REGION Network 59: Magazine Z-Axis Brake Test Error
   RUNG wire#powerrail
      { S7_Templates := "SrcType := Int" } GE_Contact(in1 := "Unit1.Em5.ControlNodes".cm.brakeTest.magazine.monitoring."step", in2 := 5)
      { S7_Templates := "SrcType := Int" } LE_Contact(in1 := "Unit1.Em5.ControlNodes".cm.brakeTest.magazine.monitoring."step", in2 := 30)
      { S7_Templates := "time_type := Time" } #statTonTimer[60].TON(pt := T#10s, et =>)
      wire#w1
      Coil( "Unit1.Em5.ControlNodes".cm.brakeTest.magazine.monitoring.error )
      R_Coil( "Unit1.Em5.ControlNodes".cm.brakeTest.magazine.monitoring.busy )
      R_Coil( "Unit1.Em5.ControlNodes".cm.brakeTest.magazine.commands.axisReset )
   END_RUNG
   RUNG wire#powerrail
      Contact( "Unit1.Em5.ControlNodes".cm.brakeTest.magazine.monitoring.error )
      I_Contact( #statUnitStatus.acknowledgeActive )
   END_RUNG wire#w1
   RUNG wire#powerrail
      Contact( "Unit1.Em5.ControlNodes".cm.brakeTest.magazine.monitoring.busy )
      wire#w2
      P_Trig( #statPulse[62] )
      S_Coil( "Unit1.Em5.Config".cmMagazineAxisZ.disableAlarms )
   END_RUNG
   RUNG wire#w2
      Not()
      P_Trig( #statPulse[63] )
      R_Coil( "Unit1.Em5.Config".cmMagazineAxisZ.disableAlarms )
   END_RUNG
   // the same network as SCL:
   #statTonTimer[60].TON(IN := ("Unit1.Em5.ControlNodes".cm.brakeTest.magazine.monitoring."step" >= 5) AND ("Unit1.Em5.ControlNodes".cm.brakeTest.magazine.monitoring."step" <= 30),
                         PT := T#10s);
   "Unit1.Em5.ControlNodes".cm.brakeTest.magazine.monitoring.error := #statTonTimer[60].Q OR ("Unit1.Em5.ControlNodes".cm.brakeTest.magazine.monitoring.error AND NOT #statUnitStatus.acknowledgeActive);
   IF "Unit1.Em5.ControlNodes".cm.brakeTest.magazine.monitoring.error THEN
       "Unit1.Em5.ControlNodes".cm.brakeTest.magazine.monitoring.busy := FALSE;
       "Unit1.Em5.ControlNodes".cm.brakeTest.magazine.commands.axisReset := FALSE;
   END_IF;
   #_w1 := "Unit1.Em5.ControlNodes".cm.brakeTest.magazine.monitoring.busy AND NOT #statPulse[62];   // rising edge
   #statPulse[62] := "Unit1.Em5.ControlNodes".cm.brakeTest.magazine.monitoring.busy;
   IF #_w1 THEN "Unit1.Em5.Config".cmMagazineAxisZ.disableAlarms := TRUE; END_IF;
   #_w2 := NOT "Unit1.Em5.ControlNodes".cm.brakeTest.magazine.monitoring.busy AND NOT #statPulse[63];   // rising edge
   #statPulse[63] := NOT "Unit1.Em5.ControlNodes".cm.brakeTest.magazine.monitoring.busy;
   IF #_w2 THEN "Unit1.Em5.Config".cmMagazineAxisZ.disableAlarms := FALSE; END_IF;
END_REGION

REGION Network 60: Magazine Z-Axis Brake Test Initialize
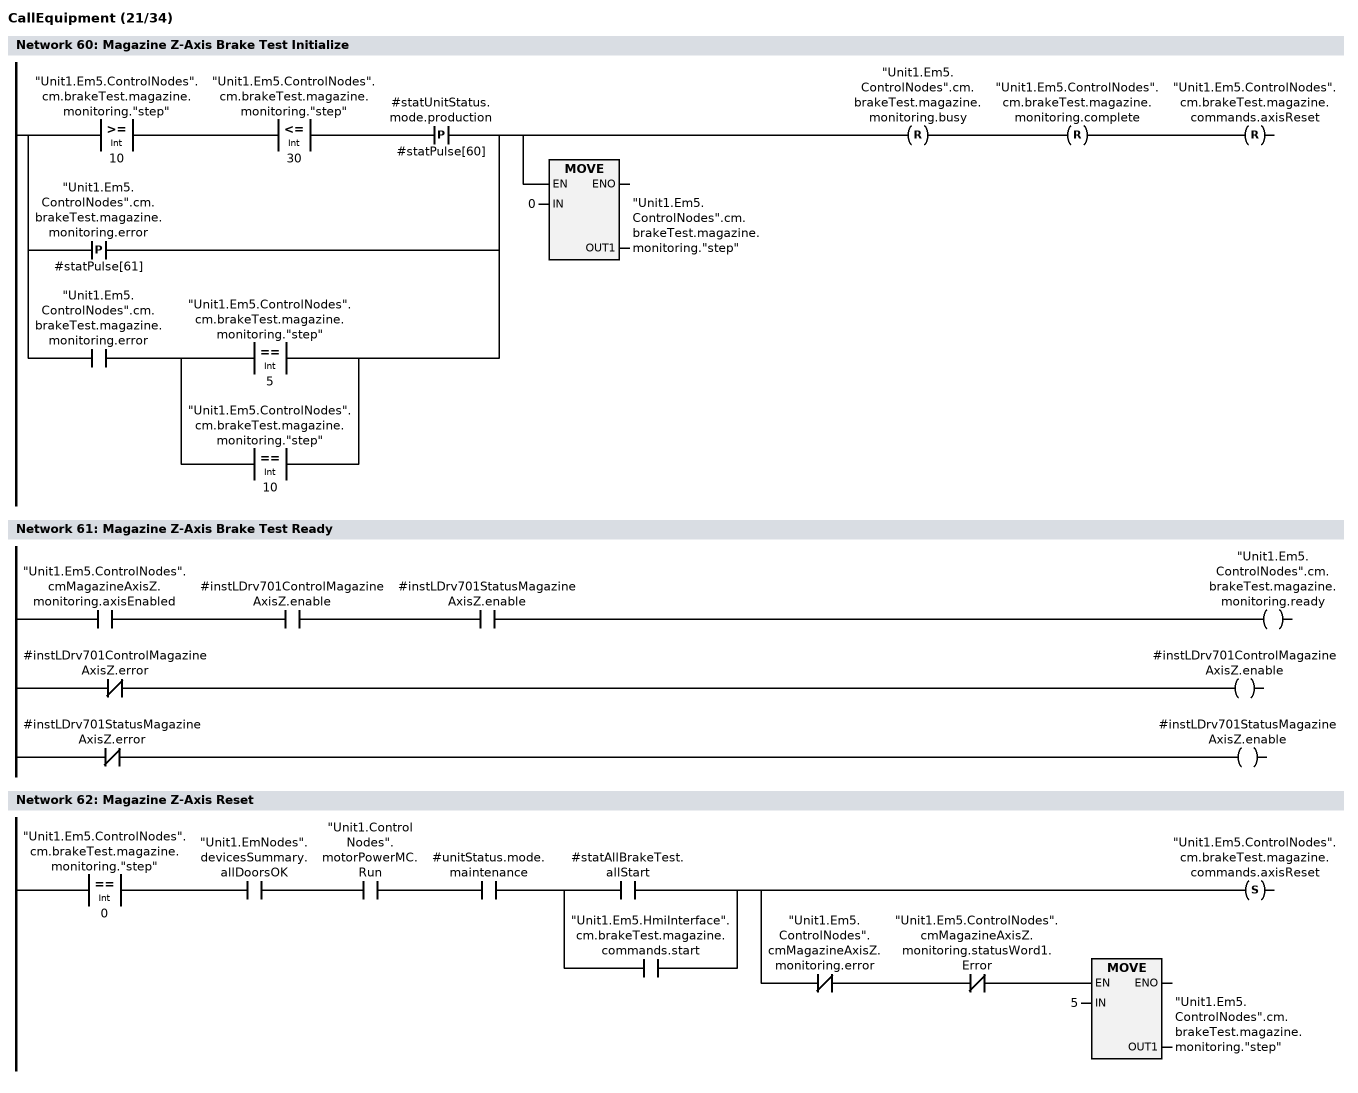
   RUNG wire#powerrail
      { S7_Templates := "SrcType := Int" } GE_Contact(in1 := "Unit1.Em5.ControlNodes".cm.brakeTest.magazine.monitoring."step", in2 := 10)
      { S7_Templates := "SrcType := Int" } LE_Contact(in1 := "Unit1.Em5.ControlNodes".cm.brakeTest.magazine.monitoring."step", in2 := 30)
      P_Contact(operand := #statUnitStatus.mode.production, bit := #statPulse[60])
      wire#w1
      R_Coil( "Unit1.Em5.ControlNodes".cm.brakeTest.magazine.monitoring.busy )
      R_Coil( "Unit1.Em5.ControlNodes".cm.brakeTest.magazine.monitoring.complete )
      R_Coil( "Unit1.Em5.ControlNodes".cm.brakeTest.magazine.commands.axisReset )
   END_RUNG
   RUNG wire#powerrail
      P_Contact(operand := "Unit1.Em5.ControlNodes".cm.brakeTest.magazine.monitoring.error, bit := #statPulse[61])
   END_RUNG wire#w1
   RUNG wire#powerrail
      Contact( "Unit1.Em5.ControlNodes".cm.brakeTest.magazine.monitoring.error )
      wire#w2
      { S7_Templates := "SrcType := Int" } EQ_Contact(in1 := "Unit1.Em5.ControlNodes".cm.brakeTest.magazine.monitoring."step", in2 := 5)
   END_RUNG wire#w1
   RUNG wire#w2
      { S7_Templates := "SrcType := Int" } EQ_Contact(in1 := "Unit1.Em5.ControlNodes".cm.brakeTest.magazine.monitoring."step", in2 := 10)
   END_RUNG wire#w1
   RUNG wire#w1
      Move(in := 0, out1 => "Unit1.Em5.ControlNodes".cm.brakeTest.magazine.monitoring."step")
   END_RUNG
   // the same network as SCL:
   #_w1 := ("Unit1.Em5.ControlNodes".cm.brakeTest.magazine.monitoring."step" >= 10) AND ("Unit1.Em5.ControlNodes".cm.brakeTest.magazine.monitoring."step" <= 30) AND #statUnitStatus.mode.production AND NOT #statPulse[60];   // rising edge of #statUnitStatus.mode.production
   #statPulse[60] := #statUnitStatus.mode.production;
   #_w2 := "Unit1.Em5.ControlNodes".cm.brakeTest.magazine.monitoring.error AND NOT #statPulse[61];   // rising edge of "Unit1.Em5.ControlNodes".cm.brakeTest.magazine.monitoring.error
   #statPulse[61] := "Unit1.Em5.ControlNodes".cm.brakeTest.magazine.monitoring.error;
   IF #_w1 OR #_w2 OR ("Unit1.Em5.ControlNodes".cm.brakeTest.magazine.monitoring.error AND (("Unit1.Em5.ControlNodes".cm.brakeTest.magazine.monitoring."step" = 5) OR ("Unit1.Em5.ControlNodes".cm.brakeTest.magazine.monitoring."step" = 10))) THEN
       "Unit1.Em5.ControlNodes".cm.brakeTest.magazine.monitoring.busy := FALSE;
       "Unit1.Em5.ControlNodes".cm.brakeTest.magazine.monitoring.complete := FALSE;
       "Unit1.Em5.ControlNodes".cm.brakeTest.magazine.commands.axisReset := FALSE;
       "Unit1.Em5.ControlNodes".cm.brakeTest.magazine.monitoring."step" := 0;
   END_IF;
END_REGION

REGION Network 61: Magazine Z-Axis Brake Test Ready
   RUNG wire#powerrail
      Contact( "Unit1.Em5.ControlNodes".cmMagazineAxisZ.monitoring.axisEnabled )
      Contact( #instLDrv701ControlMagazineAxisZ.enable )
      Contact( #instLDrv701StatusMagazineAxisZ.enable )
      Coil( "Unit1.Em5.ControlNodes".cm.brakeTest.magazine.monitoring.ready )
   END_RUNG
   RUNG wire#powerrail
      I_Contact( #instLDrv701ControlMagazineAxisZ.error )
      Coil( #instLDrv701ControlMagazineAxisZ.enable )
   END_RUNG
   RUNG wire#powerrail
      I_Contact( #instLDrv701StatusMagazineAxisZ.error )
      Coil( #instLDrv701StatusMagazineAxisZ.enable )
   END_RUNG
   // the same network as SCL:
   "Unit1.Em5.ControlNodes".cm.brakeTest.magazine.monitoring.ready := "Unit1.Em5.ControlNodes".cmMagazineAxisZ.monitoring.axisEnabled AND #instLDrv701ControlMagazineAxisZ.enable AND #instLDrv701StatusMagazineAxisZ.enable;
   #instLDrv701ControlMagazineAxisZ.enable := NOT #instLDrv701ControlMagazineAxisZ.error;
   #instLDrv701StatusMagazineAxisZ.enable := NOT #instLDrv701StatusMagazineAxisZ.error;
END_REGION

REGION Network 62: Magazine Z-Axis Reset
   RUNG wire#powerrail
      { S7_Templates := "SrcType := Int" } EQ_Contact(in1 := "Unit1.Em5.ControlNodes".cm.brakeTest.magazine.monitoring."step", in2 := 0)
      Contact( "Unit1.EmNodes".devicesSummary.allDoorsOK )
      Contact( "Unit1.ControlNodes".motorPowerMC.Run )
      Contact( #unitStatus.mode.maintenance )
      wire#w1
      Contact( #statAllBrakeTest.allStart )
      wire#w2
      S_Coil( "Unit1.Em5.ControlNodes".cm.brakeTest.magazine.commands.axisReset )
   END_RUNG
   RUNG wire#w1
      Contact( "Unit1.Em5.HmiInterface".cm.brakeTest.magazine.commands.start )
   END_RUNG wire#w2
   RUNG wire#w2
      I_Contact( "Unit1.Em5.ControlNodes".cmMagazineAxisZ.monitoring.error )
      I_Contact( "Unit1.Em5.ControlNodes".cmMagazineAxisZ.monitoring.statusWord1.Error )
      Move(in := 5, out1 => "Unit1.Em5.ControlNodes".cm.brakeTest.magazine.monitoring."step")
   END_RUNG
   // the same network as SCL:
   #_w1 := ("Unit1.Em5.ControlNodes".cm.brakeTest.magazine.monitoring."step" = 0) AND "Unit1.EmNodes".devicesSummary.allDoorsOK AND "Unit1.ControlNodes".motorPowerMC.Run AND #unitStatus.mode.maintenance AND (#statAllBrakeTest.allStart OR "Unit1.Em5.HmiInterface".cm.brakeTest.magazine.commands.start);
   IF #_w1 THEN "Unit1.Em5.ControlNodes".cm.brakeTest.magazine.commands.axisReset := TRUE; END_IF;
   IF #_w1 AND NOT "Unit1.Em5.ControlNodes".cmMagazineAxisZ.monitoring.error AND NOT "Unit1.Em5.ControlNodes".cmMagazineAxisZ.monitoring.statusWord1.Error THEN
       "Unit1.Em5.ControlNodes".cm.brakeTest.magazine.monitoring."step" := 5;
   END_IF;
END_REGION

REGION Network 63: Magazine Z-Axis Brake Test Commands
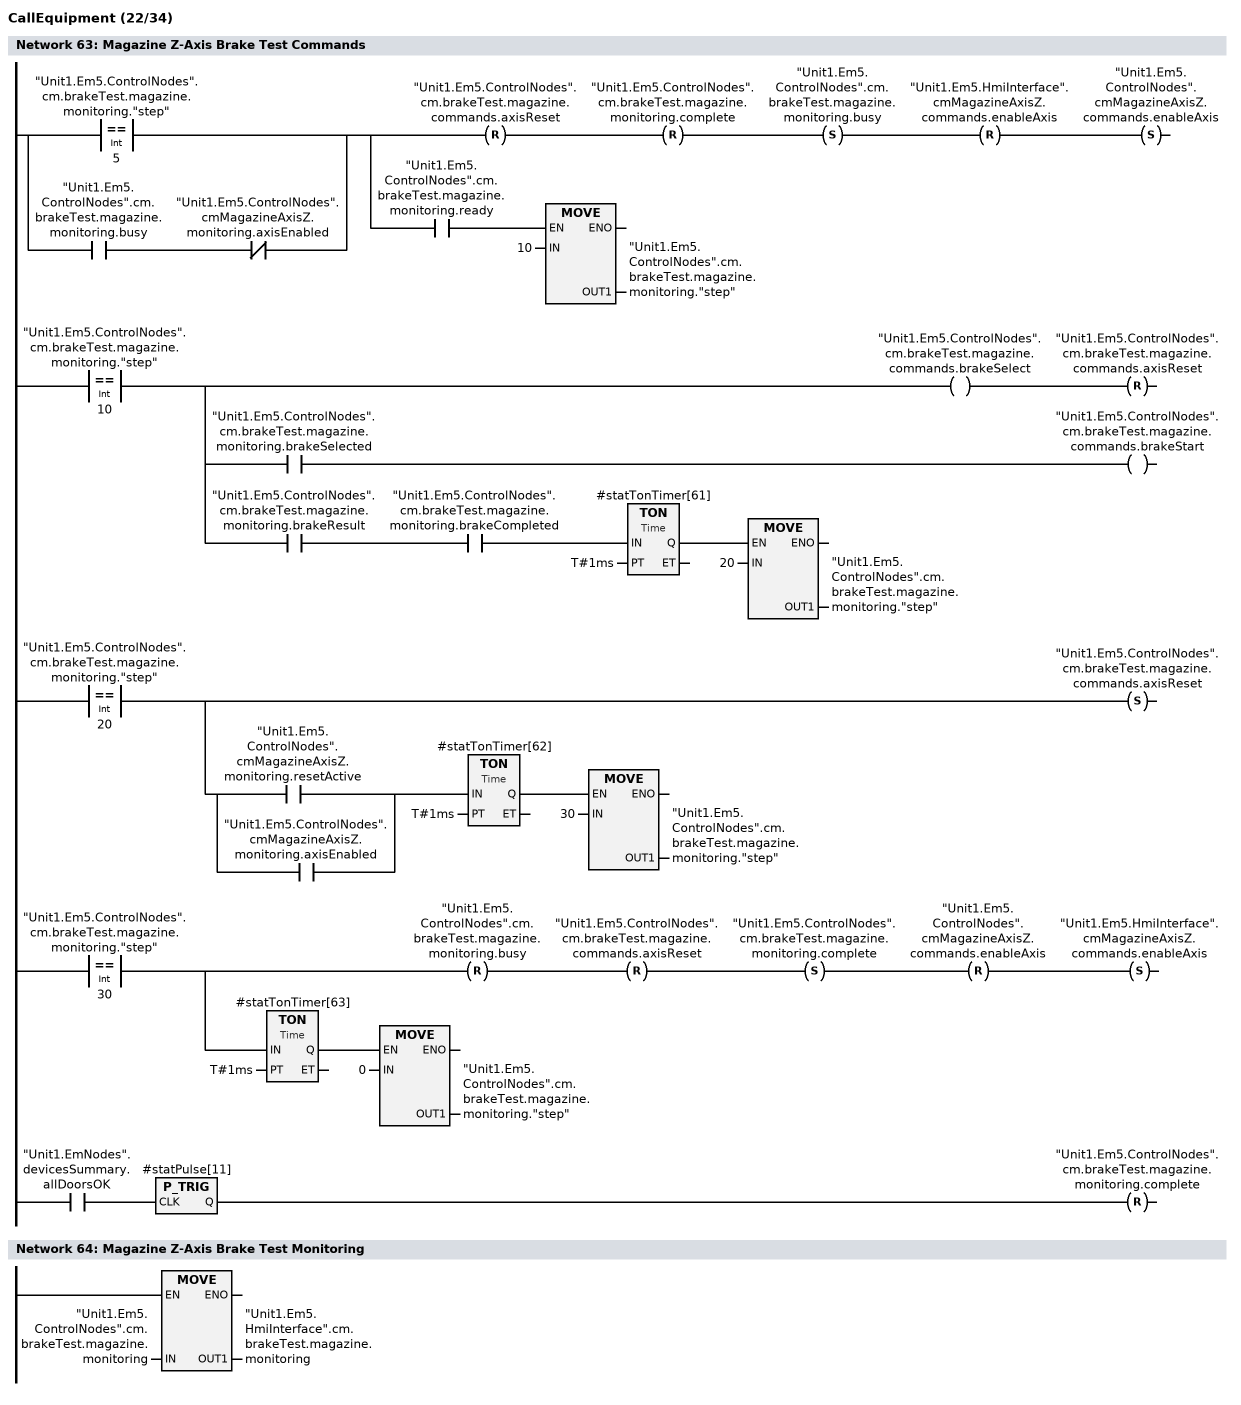
   RUNG wire#powerrail
      { S7_Templates := "SrcType := Int" } EQ_Contact(in1 := "Unit1.Em5.ControlNodes".cm.brakeTest.magazine.monitoring."step", in2 := 5)
      wire#w1
      R_Coil( "Unit1.Em5.ControlNodes".cm.brakeTest.magazine.commands.axisReset )
      R_Coil( "Unit1.Em5.ControlNodes".cm.brakeTest.magazine.monitoring.complete )
      S_Coil( "Unit1.Em5.ControlNodes".cm.brakeTest.magazine.monitoring.busy )
      R_Coil( "Unit1.Em5.HmiInterface".cmMagazineAxisZ.commands.enableAxis )
      S_Coil( "Unit1.Em5.ControlNodes".cmMagazineAxisZ.commands.enableAxis )
   END_RUNG
   RUNG wire#powerrail
      Contact( "Unit1.Em5.ControlNodes".cm.brakeTest.magazine.monitoring.busy )
      I_Contact( "Unit1.Em5.ControlNodes".cmMagazineAxisZ.monitoring.axisEnabled )
   END_RUNG wire#w1
   RUNG wire#w1
      Contact( "Unit1.Em5.ControlNodes".cm.brakeTest.magazine.monitoring.ready )
      Move(in := 10, out1 => "Unit1.Em5.ControlNodes".cm.brakeTest.magazine.monitoring."step")
   END_RUNG
   RUNG wire#powerrail
      { S7_Templates := "SrcType := Int" } EQ_Contact(in1 := "Unit1.Em5.ControlNodes".cm.brakeTest.magazine.monitoring."step", in2 := 10)
      wire#w2
      Coil( "Unit1.Em5.ControlNodes".cm.brakeTest.magazine.commands.brakeSelect )
      R_Coil( "Unit1.Em5.ControlNodes".cm.brakeTest.magazine.commands.axisReset )
   END_RUNG
   RUNG wire#w2
      Contact( "Unit1.Em5.ControlNodes".cm.brakeTest.magazine.monitoring.brakeSelected )
      Coil( "Unit1.Em5.ControlNodes".cm.brakeTest.magazine.commands.brakeStart )
   END_RUNG
   RUNG wire#w2
      Contact( "Unit1.Em5.ControlNodes".cm.brakeTest.magazine.monitoring.brakeResult )
      Contact( "Unit1.Em5.ControlNodes".cm.brakeTest.magazine.monitoring.brakeCompleted )
      { S7_Templates := "time_type := Time" } #statTonTimer[61].TON(pt := T#1ms, et =>)
      Move(in := 20, out1 => "Unit1.Em5.ControlNodes".cm.brakeTest.magazine.monitoring."step")
   END_RUNG
   RUNG wire#powerrail
      { S7_Templates := "SrcType := Int" } EQ_Contact(in1 := "Unit1.Em5.ControlNodes".cm.brakeTest.magazine.monitoring."step", in2 := 20)
      wire#w3
      S_Coil( "Unit1.Em5.ControlNodes".cm.brakeTest.magazine.commands.axisReset )
   END_RUNG
   RUNG wire#w3
      Contact( "Unit1.Em5.ControlNodes".cmMagazineAxisZ.monitoring.resetActive )
      wire#w4
      { S7_Templates := "time_type := Time" } #statTonTimer[62].TON(pt := T#1ms, et =>)
      Move(in := 30, out1 => "Unit1.Em5.ControlNodes".cm.brakeTest.magazine.monitoring."step")
   END_RUNG
   RUNG wire#w3
      Contact( "Unit1.Em5.ControlNodes".cmMagazineAxisZ.monitoring.axisEnabled )
   END_RUNG wire#w4
   RUNG wire#powerrail
      { S7_Templates := "SrcType := Int" } EQ_Contact(in1 := "Unit1.Em5.ControlNodes".cm.brakeTest.magazine.monitoring."step", in2 := 30)
      wire#w5
      R_Coil( "Unit1.Em5.ControlNodes".cm.brakeTest.magazine.monitoring.busy )
      R_Coil( "Unit1.Em5.ControlNodes".cm.brakeTest.magazine.commands.axisReset )
      S_Coil( "Unit1.Em5.ControlNodes".cm.brakeTest.magazine.monitoring.complete )
      R_Coil( "Unit1.Em5.ControlNodes".cmMagazineAxisZ.commands.enableAxis )
      S_Coil( "Unit1.Em5.HmiInterface".cmMagazineAxisZ.commands.enableAxis )
   END_RUNG
   RUNG wire#w5
      { S7_Templates := "time_type := Time" } #statTonTimer[63].TON(pt := T#1ms, et =>)
      Move(in := 0, out1 => "Unit1.Em5.ControlNodes".cm.brakeTest.magazine.monitoring."step")
   END_RUNG
   RUNG wire#powerrail
      Contact( "Unit1.EmNodes".devicesSummary.allDoorsOK )
      P_Trig( #statPulse[11] )
      R_Coil( "Unit1.Em5.ControlNodes".cm.brakeTest.magazine.monitoring.complete )
   END_RUNG
   // the same network as SCL:
   #_w1 := ("Unit1.Em5.ControlNodes".cm.brakeTest.magazine.monitoring."step" = 5) OR ("Unit1.Em5.ControlNodes".cm.brakeTest.magazine.monitoring.busy AND NOT "Unit1.Em5.ControlNodes".cmMagazineAxisZ.monitoring.axisEnabled);
   IF #_w1 THEN
       "Unit1.Em5.ControlNodes".cm.brakeTest.magazine.commands.axisReset := FALSE;
       "Unit1.Em5.ControlNodes".cm.brakeTest.magazine.monitoring.complete := FALSE;
       "Unit1.Em5.ControlNodes".cm.brakeTest.magazine.monitoring.busy := TRUE;
       "Unit1.Em5.HmiInterface".cmMagazineAxisZ.commands.enableAxis := FALSE;
       "Unit1.Em5.ControlNodes".cmMagazineAxisZ.commands.enableAxis := TRUE;
   END_IF;
   IF #_w1 AND "Unit1.Em5.ControlNodes".cm.brakeTest.magazine.monitoring.ready THEN
       "Unit1.Em5.ControlNodes".cm.brakeTest.magazine.monitoring."step" := 10;
   END_IF;
   "Unit1.Em5.ControlNodes".cm.brakeTest.magazine.commands.brakeSelect := "Unit1.Em5.ControlNodes".cm.brakeTest.magazine.monitoring."step" = 10;
   IF "Unit1.Em5.ControlNodes".cm.brakeTest.magazine.commands.brakeSelect THEN
       "Unit1.Em5.ControlNodes".cm.brakeTest.magazine.commands.axisReset := FALSE;
   END_IF;
   "Unit1.Em5.ControlNodes".cm.brakeTest.magazine.commands.brakeStart := "Unit1.Em5.ControlNodes".cm.brakeTest.magazine.commands.brakeSelect AND "Unit1.Em5.ControlNodes".cm.brakeTest.magazine.monitoring.brakeSelected;
   #statTonTimer[61].TON(IN := "Unit1.Em5.ControlNodes".cm.brakeTest.magazine.commands.brakeSelect AND "Unit1.Em5.ControlNodes".cm.brakeTest.magazine.monitoring.brakeResult AND "Unit1.Em5.ControlNodes".cm.brakeTest.magazine.monitoring.brakeCompleted,
                         PT := T#1ms);
   IF #statTonTimer[61].Q THEN
       "Unit1.Em5.ControlNodes".cm.brakeTest.magazine.monitoring."step" := 20;
   END_IF;
   #_w2 := "Unit1.Em5.ControlNodes".cm.brakeTest.magazine.monitoring."step" = 20;
   IF #_w2 THEN "Unit1.Em5.ControlNodes".cm.brakeTest.magazine.commands.axisReset := TRUE; END_IF;
   #statTonTimer[62].TON(IN := #_w2 AND ("Unit1.Em5.ControlNodes".cmMagazineAxisZ.monitoring.resetActive OR "Unit1.Em5.ControlNodes".cmMagazineAxisZ.monitoring.axisEnabled),
                         PT := T#1ms);
   IF #statTonTimer[62].Q THEN
       "Unit1.Em5.ControlNodes".cm.brakeTest.magazine.monitoring."step" := 30;
   END_IF;
   #_w3 := "Unit1.Em5.ControlNodes".cm.brakeTest.magazine.monitoring."step" = 30;
   IF #_w3 THEN
       "Unit1.Em5.ControlNodes".cm.brakeTest.magazine.monitoring.busy := FALSE;
       "Unit1.Em5.ControlNodes".cm.brakeTest.magazine.commands.axisReset := FALSE;
       "Unit1.Em5.ControlNodes".cm.brakeTest.magazine.monitoring.complete := TRUE;
       "Unit1.Em5.ControlNodes".cmMagazineAxisZ.commands.enableAxis := FALSE;
       "Unit1.Em5.HmiInterface".cmMagazineAxisZ.commands.enableAxis := TRUE;
   END_IF;
   #statTonTimer[63].TON(IN := #_w3, PT := T#1ms);
   IF #statTonTimer[63].Q THEN "Unit1.Em5.ControlNodes".cm.brakeTest.magazine.monitoring."step" := 0; END_IF;
   #_w4 := "Unit1.EmNodes".devicesSummary.allDoorsOK AND NOT #statPulse[11];   // rising edge
   #statPulse[11] := "Unit1.EmNodes".devicesSummary.allDoorsOK;
   IF #_w4 THEN "Unit1.Em5.ControlNodes".cm.brakeTest.magazine.monitoring.complete := FALSE; END_IF;
END_REGION

REGION Network 64: Magazine Z-Axis Brake Test Monitoring
   RUNG wire#powerrail
      Move(in := "Unit1.Em5.ControlNodes".cm.brakeTest.magazine.monitoring, out1 => "Unit1.Em5.HmiInterface".cm.brakeTest.magazine.monitoring)
   END_RUNG
   // the same network as SCL:
   "Unit1.Em5.HmiInterface".cm.brakeTest.magazine.monitoring := "Unit1.Em5.ControlNodes".cm.brakeTest.magazine.monitoring;
END_REGION

REGION Network 65: Call Magazine Z-Axis Telegram 701
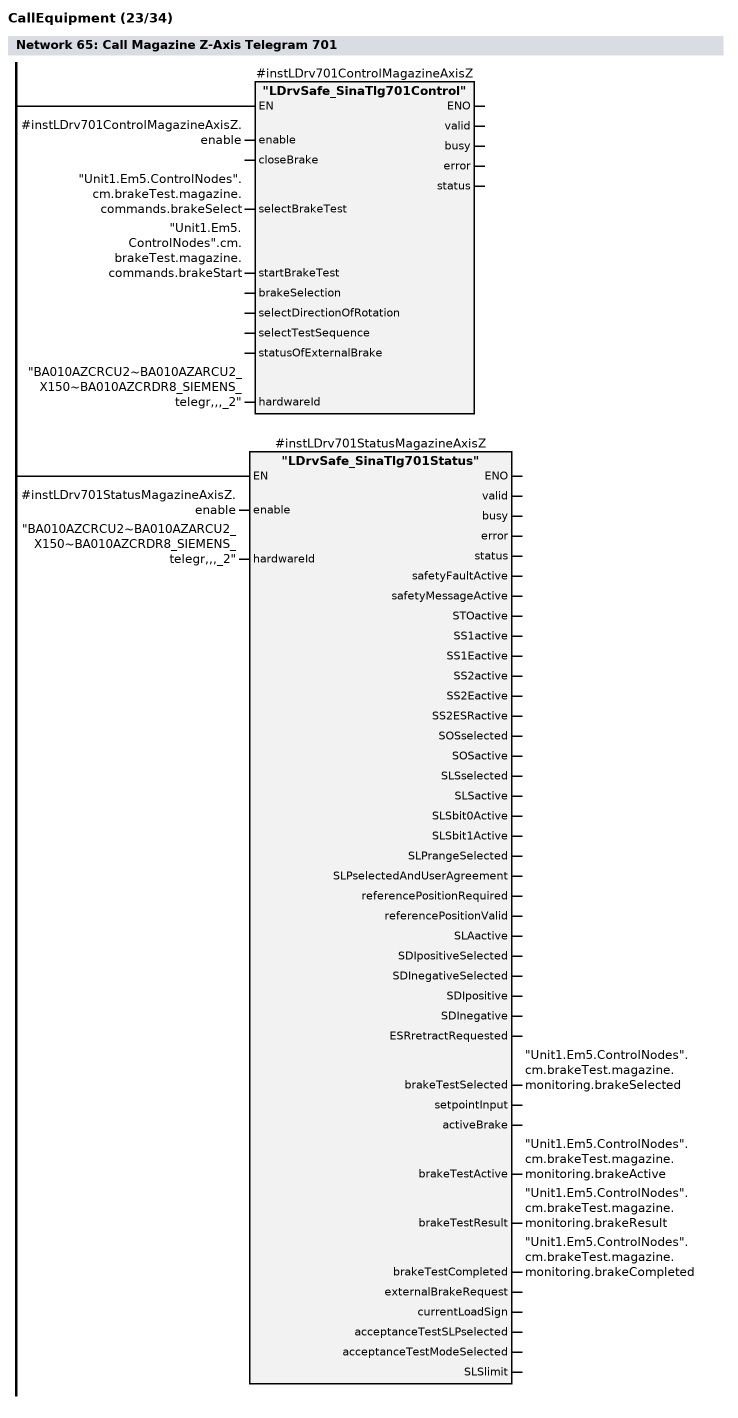
   RUNG wire#powerrail
      #instLDrv701ControlMagazineAxisZ(enable := #instLDrv701ControlMagazineAxisZ.enable, closeBrake :=, selectBrakeTest := "Unit1.Em5.ControlNodes".cm.brakeTest.magazine.commands.brakeSelect, startBrakeTest := "Unit1.Em5.ControlNodes".cm.brakeTest.magazine.commands.brakeStart, brakeSelection :=, selectDirectionOfRotation :=, selectTestSequence :=, statusOfExternalBrake :=, hardwareId := "BA010AZCRCU2~BA010AZARCU2_X150~BA010AZCRDR8_SIEMENS_telegr,,,_2", valid =>, busy =>, error =>, status =>)
   END_RUNG
   RUNG wire#powerrail
      #instLDrv701StatusMagazineAxisZ(enable := #instLDrv701StatusMagazineAxisZ.enable, hardwareId := "BA010AZCRCU2~BA010AZARCU2_X150~BA010AZCRDR8_SIEMENS_telegr,,,_2", valid =>, busy =>, error =>, status =>, safetyFaultActive =>, safetyMessageActive =>, STOactive =>, SS1active =>, SS1Eactive =>, SS2active =>, SS2Eactive =>, SS2ESRactive =>, SOSselected =>, SOSactive =>, SLSselected =>, SLSactive =>, SLSbit0Active =>, SLSbit1Active =>, SLPrangeSelected =>, SLPselectedAndUserAgreement =>, referencePositionRequired =>, referencePositionValid =>, SLAactive =>, SDIpositiveSelected =>, SDInegativeSelected =>, SDIpositive =>, SDInegative =>, ESRretractRequested =>, brakeTestSelected => "Unit1.Em5.ControlNodes".cm.brakeTest.magazine.monitoring.brakeSelected, setpointInput =>, activeBrake =>, brakeTestActive => "Unit1.Em5.ControlNodes".cm.brakeTest.magazine.monitoring.brakeActive, brakeTestResult => "Unit1.Em5.ControlNodes".cm.brakeTest.magazine.monitoring.brakeResult, brakeTestCompleted => "Unit1.Em5.ControlNodes".cm.brakeTest.magazine.monitoring.brakeCompleted, externalBrakeRequest =>, currentLoadSign =>, acceptanceTestSLPselected =>, acceptanceTestModeSelected =>, SLSlimit =>)
   END_RUNG
   // the same network as SCL:
   #instLDrv701ControlMagazineAxisZ(enable := #instLDrv701ControlMagazineAxisZ.enable,   // "LDrvSafe_SinaTlg701Control"
                           selectBrakeTest := "Unit1.Em5.ControlNodes".cm.brakeTest.magazine.commands.brakeSelect,
                           startBrakeTest := "Unit1.Em5.ControlNodes".cm.brakeTest.magazine.commands.brakeStart,
                           hardwareId := "BA010AZCRCU2~BA010AZARCU2_X150~BA010AZCRDR8_SIEMENS_telegr,,,_2");
   #instLDrv701StatusMagazineAxisZ(enable := #instLDrv701StatusMagazineAxisZ.enable,   // "LDrvSafe_SinaTlg701Status"
                           hardwareId := "BA010AZCRCU2~BA010AZARCU2_X150~BA010AZCRDR8_SIEMENS_telegr,,,_2",
                           brakeTestSelected => "Unit1.Em5.ControlNodes".cm.brakeTest.magazine.monitoring.brakeSelected,
                           brakeTestActive => "Unit1.Em5.ControlNodes".cm.brakeTest.magazine.monitoring.brakeActive,
                           brakeTestResult => "Unit1.Em5.ControlNodes".cm.brakeTest.magazine.monitoring.brakeResult,
                           brakeTestCompleted => "Unit1.Em5.ControlNodes".cm.brakeTest.magazine.monitoring.brakeCompleted);
END_REGION

REGION Network 67: ******************** Control Modules (TwoWayActuator) ********************
   // Call control modules that are actuators after the em logic (jobs and sequence), so that the latest commands are applied to the actuators.
END_REGION

REGION Network 68: Reset CMS
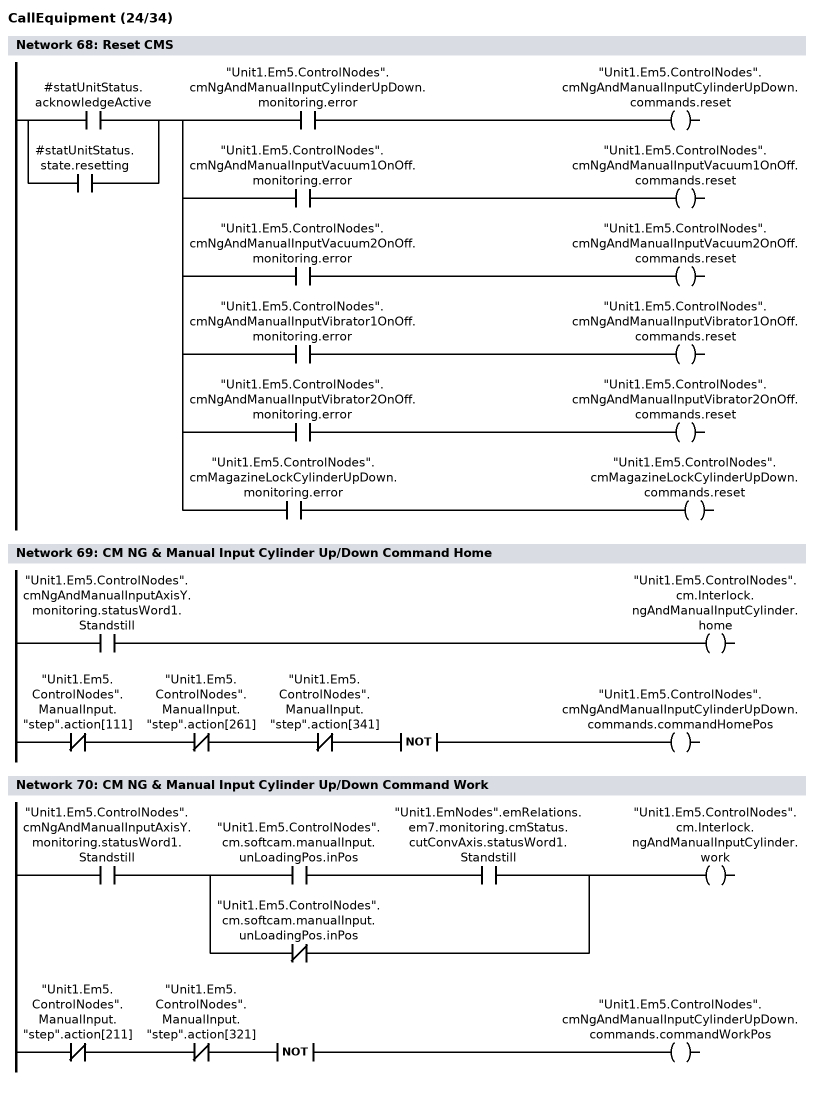
   RUNG wire#powerrail
      Contact( #statUnitStatus.acknowledgeActive )
      wire#w1
      Contact( "Unit1.Em5.ControlNodes".cmNgAndManualInputCylinderUpDown.monitoring.error )
      Coil( "Unit1.Em5.ControlNodes".cmNgAndManualInputCylinderUpDown.commands.reset )
   END_RUNG
   RUNG wire#powerrail
      Contact( #statUnitStatus.state.resetting )
   END_RUNG wire#w1
   RUNG wire#w1
      Contact( "Unit1.Em5.ControlNodes".cmNgAndManualInputVacuum1OnOff.monitoring.error )
      Coil( "Unit1.Em5.ControlNodes".cmNgAndManualInputVacuum1OnOff.commands.reset )
   END_RUNG
   RUNG wire#w1
      Contact( "Unit1.Em5.ControlNodes".cmNgAndManualInputVacuum2OnOff.monitoring.error )
      Coil( "Unit1.Em5.ControlNodes".cmNgAndManualInputVacuum2OnOff.commands.reset )
   END_RUNG
   RUNG wire#w1
      Contact( "Unit1.Em5.ControlNodes".cmNgAndManualInputVibrator1OnOff.monitoring.error )
      Coil( "Unit1.Em5.ControlNodes".cmNgAndManualInputVibrator1OnOff.commands.reset )
   END_RUNG
   RUNG wire#w1
      Contact( "Unit1.Em5.ControlNodes".cmNgAndManualInputVibrator2OnOff.monitoring.error )
      Coil( "Unit1.Em5.ControlNodes".cmNgAndManualInputVibrator2OnOff.commands.reset )
   END_RUNG
   RUNG wire#w1
      Contact( "Unit1.Em5.ControlNodes".cmMagazineLockCylinderUpDown.monitoring.error )
      Coil( "Unit1.Em5.ControlNodes".cmMagazineLockCylinderUpDown.commands.reset )
   END_RUNG
   // the same network as SCL:
   #_w1 := #statUnitStatus.acknowledgeActive OR #statUnitStatus.state.resetting;
   "Unit1.Em5.ControlNodes".cmNgAndManualInputCylinderUpDown.commands.reset := #_w1 AND "Unit1.Em5.ControlNodes".cmNgAndManualInputCylinderUpDown.monitoring.error;
   "Unit1.Em5.ControlNodes".cmNgAndManualInputVacuum1OnOff.commands.reset := #_w1 AND "Unit1.Em5.ControlNodes".cmNgAndManualInputVacuum1OnOff.monitoring.error;
   "Unit1.Em5.ControlNodes".cmNgAndManualInputVacuum2OnOff.commands.reset := #_w1 AND "Unit1.Em5.ControlNodes".cmNgAndManualInputVacuum2OnOff.monitoring.error;
   "Unit1.Em5.ControlNodes".cmNgAndManualInputVibrator1OnOff.commands.reset := #_w1 AND "Unit1.Em5.ControlNodes".cmNgAndManualInputVibrator1OnOff.monitoring.error;
   "Unit1.Em5.ControlNodes".cmNgAndManualInputVibrator2OnOff.commands.reset := #_w1 AND "Unit1.Em5.ControlNodes".cmNgAndManualInputVibrator2OnOff.monitoring.error;
   "Unit1.Em5.ControlNodes".cmMagazineLockCylinderUpDown.commands.reset := #_w1 AND "Unit1.Em5.ControlNodes".cmMagazineLockCylinderUpDown.monitoring.error;
END_REGION

REGION Network 69: CM NG & Manual Input Cylinder Up/Down Command Home
   RUNG wire#powerrail
      Contact( "Unit1.Em5.ControlNodes".cmNgAndManualInputAxisY.monitoring.statusWord1.Standstill )
      Coil( "Unit1.Em5.ControlNodes".cm.Interlock.ngAndManualInputCylinder.home )
   END_RUNG
   RUNG wire#powerrail
      I_Contact( "Unit1.Em5.ControlNodes".ManualInput."step".action[111] )
      I_Contact( "Unit1.Em5.ControlNodes".ManualInput."step".action[261] )
      I_Contact( "Unit1.Em5.ControlNodes".ManualInput."step".action[341] )
      Not()
      Coil( "Unit1.Em5.ControlNodes".cmNgAndManualInputCylinderUpDown.commands.commandHomePos )
   END_RUNG
   // the same network as SCL:
   "Unit1.Em5.ControlNodes".cm.Interlock.ngAndManualInputCylinder.home := "Unit1.Em5.ControlNodes".cmNgAndManualInputAxisY.monitoring.statusWord1.Standstill;
   "Unit1.Em5.ControlNodes".cmNgAndManualInputCylinderUpDown.commands.commandHomePos := NOT (NOT "Unit1.Em5.ControlNodes".ManualInput."step".action[111] AND NOT "Unit1.Em5.ControlNodes".ManualInput."step".action[261] AND NOT "Unit1.Em5.ControlNodes".ManualInput."step".action[341]);
END_REGION

REGION Network 70: CM NG & Manual Input Cylinder Up/Down Command Work
   RUNG wire#powerrail
      Contact( "Unit1.Em5.ControlNodes".cmNgAndManualInputAxisY.monitoring.statusWord1.Standstill )
      wire#w1
      Contact( "Unit1.Em5.ControlNodes".cm.softcam.manualInput.unLoadingPos.inPos )
      Contact( "Unit1.EmNodes".emRelations.em7.monitoring.cmStatus.cutConvAxis.statusWord1.Standstill )
      wire#w2
      Coil( "Unit1.Em5.ControlNodes".cm.Interlock.ngAndManualInputCylinder.work )
   END_RUNG
   RUNG wire#w1
      I_Contact( "Unit1.Em5.ControlNodes".cm.softcam.manualInput.unLoadingPos.inPos )
   END_RUNG wire#w2
   RUNG wire#powerrail
      I_Contact( "Unit1.Em5.ControlNodes".ManualInput."step".action[211] )
      I_Contact( "Unit1.Em5.ControlNodes".ManualInput."step".action[321] )
      Not()
      Coil( "Unit1.Em5.ControlNodes".cmNgAndManualInputCylinderUpDown.commands.commandWorkPos )
   END_RUNG
   // the same network as SCL:
   "Unit1.Em5.ControlNodes".cm.Interlock.ngAndManualInputCylinder.work := "Unit1.Em5.ControlNodes".cmNgAndManualInputAxisY.monitoring.statusWord1.Standstill AND (("Unit1.Em5.ControlNodes".cm.softcam.manualInput.unLoadingPos.inPos AND "Unit1.EmNodes".emRelations.em7.monitoring.cmStatus.cutConvAxis.statusWord1.Standstill) OR NOT "Unit1.Em5.ControlNodes".cm.softcam.manualInput.unLoadingPos.inPos);
   "Unit1.Em5.ControlNodes".cmNgAndManualInputCylinderUpDown.commands.commandWorkPos := NOT (NOT "Unit1.Em5.ControlNodes".ManualInput."step".action[211] AND NOT "Unit1.Em5.ControlNodes".ManualInput."step".action[321]);
END_REGION

REGION Network 71: Call CM NG & Manual Input Cylinder Up/Down (LBC_TwoWayActuator)
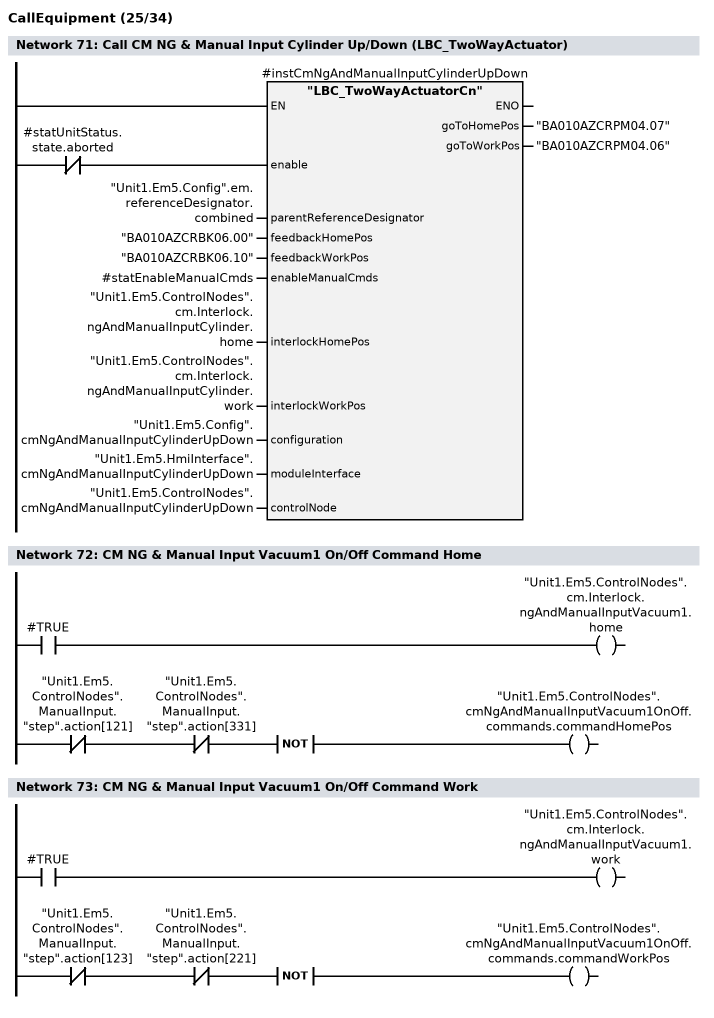
   RUNG wire#powerrail
      #instCmNgAndManualInputCylinderUpDown(enable := wire#w1, parentReferenceDesignator := "Unit1.Em5.Config".em.referenceDesignator.combined, feedbackHomePos := "BA010AZCRBK06.00", feedbackWorkPos := "BA010AZCRBK06.10", enableManualCmds := #statEnableManualCmds, interlockHomePos := "Unit1.Em5.ControlNodes".cm.Interlock.ngAndManualInputCylinder.home, interlockWorkPos := "Unit1.Em5.ControlNodes".cm.Interlock.ngAndManualInputCylinder.work, configuration := "Unit1.Em5.Config".cmNgAndManualInputCylinderUpDown, moduleInterface := "Unit1.Em5.HmiInterface".cmNgAndManualInputCylinderUpDown, controlNode := "Unit1.Em5.ControlNodes".cmNgAndManualInputCylinderUpDown, goToHomePos => "BA010AZCRPM04.07", goToWorkPos => "BA010AZCRPM04.06")
   END_RUNG
   RUNG wire#powerrail
      I_Contact( #statUnitStatus.state.aborted )
   END_RUNG wire#w1
   // the same network as SCL:
   #instCmNgAndManualInputCylinderUpDown(enable := NOT #statUnitStatus.state.aborted,   // "LBC_TwoWayActuatorCn"
                           parentReferenceDesignator := "Unit1.Em5.Config".em.referenceDesignator.combined,
                           feedbackHomePos := "BA010AZCRBK06.00",
                           feedbackWorkPos := "BA010AZCRBK06.10",
                           enableManualCmds := #statEnableManualCmds,
                           interlockHomePos := "Unit1.Em5.ControlNodes".cm.Interlock.ngAndManualInputCylinder.home,
                           interlockWorkPos := "Unit1.Em5.ControlNodes".cm.Interlock.ngAndManualInputCylinder.work,
                           configuration := "Unit1.Em5.Config".cmNgAndManualInputCylinderUpDown,
                           moduleInterface := "Unit1.Em5.HmiInterface".cmNgAndManualInputCylinderUpDown,
                           controlNode := "Unit1.Em5.ControlNodes".cmNgAndManualInputCylinderUpDown,
                           goToHomePos => "BA010AZCRPM04.07",
                           goToWorkPos => "BA010AZCRPM04.06");
END_REGION

REGION Network 72: CM NG & Manual Input Vacuum1 On/Off Command Home
   RUNG wire#powerrail
      Contact( #TRUE )
      Coil( "Unit1.Em5.ControlNodes".cm.Interlock.ngAndManualInputVacuum1.home )
   END_RUNG
   RUNG wire#powerrail
      I_Contact( "Unit1.Em5.ControlNodes".ManualInput."step".action[121] )
      I_Contact( "Unit1.Em5.ControlNodes".ManualInput."step".action[331] )
      Not()
      Coil( "Unit1.Em5.ControlNodes".cmNgAndManualInputVacuum1OnOff.commands.commandHomePos )
   END_RUNG
   // the same network as SCL:
   "Unit1.Em5.ControlNodes".cm.Interlock.ngAndManualInputVacuum1.home := #TRUE;
   "Unit1.Em5.ControlNodes".cmNgAndManualInputVacuum1OnOff.commands.commandHomePos := NOT (NOT "Unit1.Em5.ControlNodes".ManualInput."step".action[121] AND NOT "Unit1.Em5.ControlNodes".ManualInput."step".action[331]);
END_REGION

REGION Network 73: CM NG & Manual Input Vacuum1 On/Off Command Work
   RUNG wire#powerrail
      Contact( #TRUE )
      Coil( "Unit1.Em5.ControlNodes".cm.Interlock.ngAndManualInputVacuum1.work )
   END_RUNG
   RUNG wire#powerrail
      I_Contact( "Unit1.Em5.ControlNodes".ManualInput."step".action[123] )
      I_Contact( "Unit1.Em5.ControlNodes".ManualInput."step".action[221] )
      Not()
      Coil( "Unit1.Em5.ControlNodes".cmNgAndManualInputVacuum1OnOff.commands.commandWorkPos )
   END_RUNG
   // the same network as SCL:
   "Unit1.Em5.ControlNodes".cm.Interlock.ngAndManualInputVacuum1.work := #TRUE;
   "Unit1.Em5.ControlNodes".cmNgAndManualInputVacuum1OnOff.commands.commandWorkPos := NOT (NOT "Unit1.Em5.ControlNodes".ManualInput."step".action[123] AND NOT "Unit1.Em5.ControlNodes".ManualInput."step".action[221]);
END_REGION

REGION Network 74: Call CM NG & Manual Input Vacuum1 On/Off (LBC_TwoWayActuator)
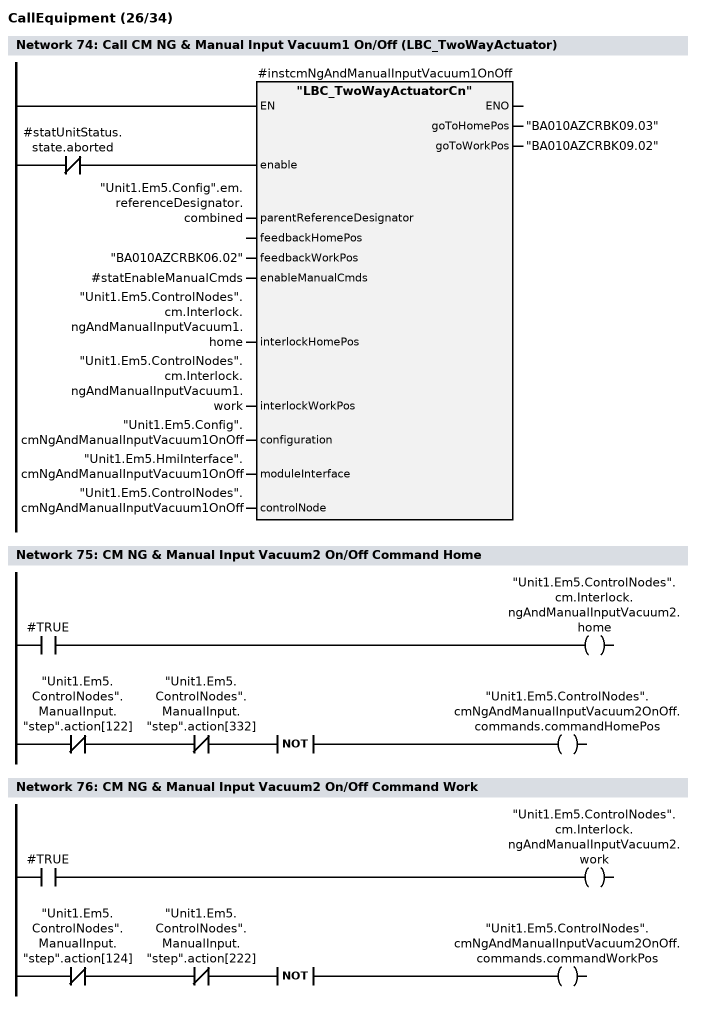
   RUNG wire#powerrail
      #instcmNgAndManualInputVacuum1OnOff(enable := wire#w1, parentReferenceDesignator := "Unit1.Em5.Config".em.referenceDesignator.combined, feedbackHomePos :=, feedbackWorkPos := "BA010AZCRBK06.02", enableManualCmds := #statEnableManualCmds, interlockHomePos := "Unit1.Em5.ControlNodes".cm.Interlock.ngAndManualInputVacuum1.home, interlockWorkPos := "Unit1.Em5.ControlNodes".cm.Interlock.ngAndManualInputVacuum1.work, configuration := "Unit1.Em5.Config".cmNgAndManualInputVacuum1OnOff, moduleInterface := "Unit1.Em5.HmiInterface".cmNgAndManualInputVacuum1OnOff, controlNode := "Unit1.Em5.ControlNodes".cmNgAndManualInputVacuum1OnOff, goToHomePos => "BA010AZCRBK09.03", goToWorkPos => "BA010AZCRBK09.02")
   END_RUNG
   RUNG wire#powerrail
      I_Contact( #statUnitStatus.state.aborted )
   END_RUNG wire#w1
   // the same network as SCL:
   #instcmNgAndManualInputVacuum1OnOff(enable := NOT #statUnitStatus.state.aborted,   // "LBC_TwoWayActuatorCn"
                           parentReferenceDesignator := "Unit1.Em5.Config".em.referenceDesignator.combined,
                           feedbackWorkPos := "BA010AZCRBK06.02",
                           enableManualCmds := #statEnableManualCmds,
                           interlockHomePos := "Unit1.Em5.ControlNodes".cm.Interlock.ngAndManualInputVacuum1.home,
                           interlockWorkPos := "Unit1.Em5.ControlNodes".cm.Interlock.ngAndManualInputVacuum1.work,
                           configuration := "Unit1.Em5.Config".cmNgAndManualInputVacuum1OnOff,
                           moduleInterface := "Unit1.Em5.HmiInterface".cmNgAndManualInputVacuum1OnOff,
                           controlNode := "Unit1.Em5.ControlNodes".cmNgAndManualInputVacuum1OnOff,
                           goToHomePos => "BA010AZCRBK09.03",
                           goToWorkPos => "BA010AZCRBK09.02");
END_REGION

REGION Network 75: CM NG & Manual Input Vacuum2 On/Off Command Home
   RUNG wire#powerrail
      Contact( #TRUE )
      Coil( "Unit1.Em5.ControlNodes".cm.Interlock.ngAndManualInputVacuum2.home )
   END_RUNG
   RUNG wire#powerrail
      I_Contact( "Unit1.Em5.ControlNodes".ManualInput."step".action[122] )
      I_Contact( "Unit1.Em5.ControlNodes".ManualInput."step".action[332] )
      Not()
      Coil( "Unit1.Em5.ControlNodes".cmNgAndManualInputVacuum2OnOff.commands.commandHomePos )
   END_RUNG
   // the same network as SCL:
   "Unit1.Em5.ControlNodes".cm.Interlock.ngAndManualInputVacuum2.home := #TRUE;
   "Unit1.Em5.ControlNodes".cmNgAndManualInputVacuum2OnOff.commands.commandHomePos := NOT (NOT "Unit1.Em5.ControlNodes".ManualInput."step".action[122] AND NOT "Unit1.Em5.ControlNodes".ManualInput."step".action[332]);
END_REGION

REGION Network 76: CM NG & Manual Input Vacuum2 On/Off Command Work
   RUNG wire#powerrail
      Contact( #TRUE )
      Coil( "Unit1.Em5.ControlNodes".cm.Interlock.ngAndManualInputVacuum2.work )
   END_RUNG
   RUNG wire#powerrail
      I_Contact( "Unit1.Em5.ControlNodes".ManualInput."step".action[124] )
      I_Contact( "Unit1.Em5.ControlNodes".ManualInput."step".action[222] )
      Not()
      Coil( "Unit1.Em5.ControlNodes".cmNgAndManualInputVacuum2OnOff.commands.commandWorkPos )
   END_RUNG
   // the same network as SCL:
   "Unit1.Em5.ControlNodes".cm.Interlock.ngAndManualInputVacuum2.work := #TRUE;
   "Unit1.Em5.ControlNodes".cmNgAndManualInputVacuum2OnOff.commands.commandWorkPos := NOT (NOT "Unit1.Em5.ControlNodes".ManualInput."step".action[124] AND NOT "Unit1.Em5.ControlNodes".ManualInput."step".action[222]);
END_REGION

REGION Network 77: Call CM NG & Manual Input Vacuum2 On/Off (LBC_TwoWayActuator)
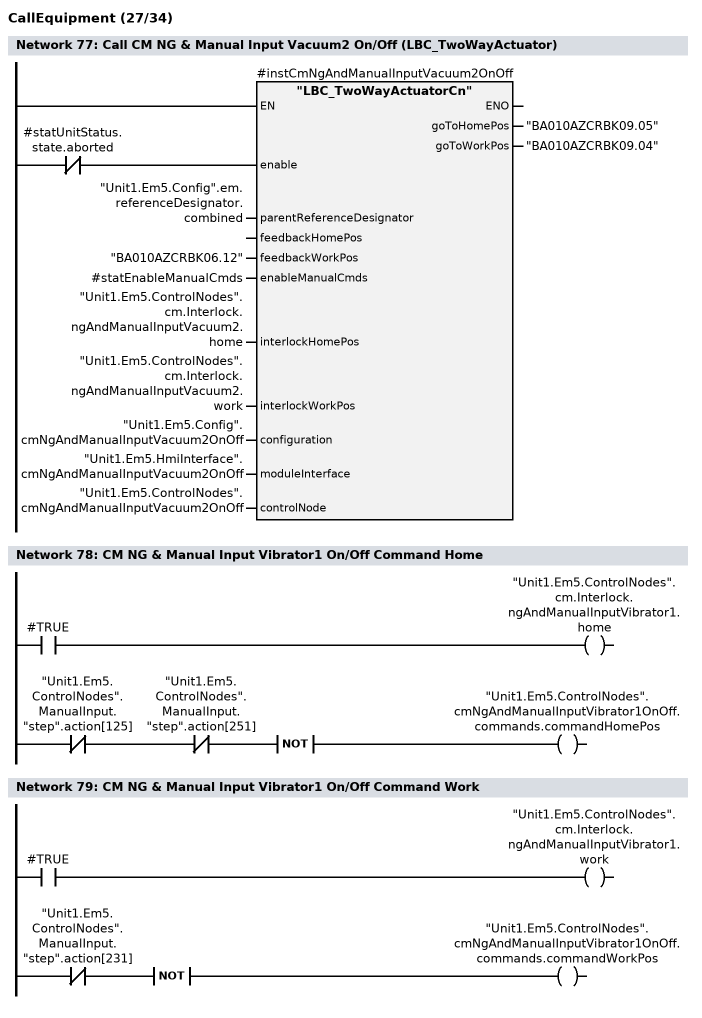
   RUNG wire#powerrail
      #instCmNgAndManualInputVacuum2OnOff(enable := wire#w1, parentReferenceDesignator := "Unit1.Em5.Config".em.referenceDesignator.combined, feedbackHomePos :=, feedbackWorkPos := "BA010AZCRBK06.12", enableManualCmds := #statEnableManualCmds, interlockHomePos := "Unit1.Em5.ControlNodes".cm.Interlock.ngAndManualInputVacuum2.home, interlockWorkPos := "Unit1.Em5.ControlNodes".cm.Interlock.ngAndManualInputVacuum2.work, configuration := "Unit1.Em5.Config".cmNgAndManualInputVacuum2OnOff, moduleInterface := "Unit1.Em5.HmiInterface".cmNgAndManualInputVacuum2OnOff, controlNode := "Unit1.Em5.ControlNodes".cmNgAndManualInputVacuum2OnOff, goToHomePos => "BA010AZCRBK09.05", goToWorkPos => "BA010AZCRBK09.04")
   END_RUNG
   RUNG wire#powerrail
      I_Contact( #statUnitStatus.state.aborted )
   END_RUNG wire#w1
   // the same network as SCL:
   #instCmNgAndManualInputVacuum2OnOff(enable := NOT #statUnitStatus.state.aborted,   // "LBC_TwoWayActuatorCn"
                           parentReferenceDesignator := "Unit1.Em5.Config".em.referenceDesignator.combined,
                           feedbackWorkPos := "BA010AZCRBK06.12",
                           enableManualCmds := #statEnableManualCmds,
                           interlockHomePos := "Unit1.Em5.ControlNodes".cm.Interlock.ngAndManualInputVacuum2.home,
                           interlockWorkPos := "Unit1.Em5.ControlNodes".cm.Interlock.ngAndManualInputVacuum2.work,
                           configuration := "Unit1.Em5.Config".cmNgAndManualInputVacuum2OnOff,
                           moduleInterface := "Unit1.Em5.HmiInterface".cmNgAndManualInputVacuum2OnOff,
                           controlNode := "Unit1.Em5.ControlNodes".cmNgAndManualInputVacuum2OnOff,
                           goToHomePos => "BA010AZCRBK09.05",
                           goToWorkPos => "BA010AZCRBK09.04");
END_REGION

REGION Network 78: CM NG & Manual Input Vibrator1 On/Off Command Home
   RUNG wire#powerrail
      Contact( #TRUE )
      Coil( "Unit1.Em5.ControlNodes".cm.Interlock.ngAndManualInputVibrator1.home )
   END_RUNG
   RUNG wire#powerrail
      I_Contact( "Unit1.Em5.ControlNodes".ManualInput."step".action[125] )
      I_Contact( "Unit1.Em5.ControlNodes".ManualInput."step".action[251] )
      Not()
      Coil( "Unit1.Em5.ControlNodes".cmNgAndManualInputVibrator1OnOff.commands.commandHomePos )
   END_RUNG
   // the same network as SCL:
   "Unit1.Em5.ControlNodes".cm.Interlock.ngAndManualInputVibrator1.home := #TRUE;
   "Unit1.Em5.ControlNodes".cmNgAndManualInputVibrator1OnOff.commands.commandHomePos := NOT (NOT "Unit1.Em5.ControlNodes".ManualInput."step".action[125] AND NOT "Unit1.Em5.ControlNodes".ManualInput."step".action[251]);
END_REGION

REGION Network 79: CM NG & Manual Input Vibrator1 On/Off Command Work
   RUNG wire#powerrail
      Contact( #TRUE )
      Coil( "Unit1.Em5.ControlNodes".cm.Interlock.ngAndManualInputVibrator1.work )
   END_RUNG
   RUNG wire#powerrail
      I_Contact( "Unit1.Em5.ControlNodes".ManualInput."step".action[231] )
      Not()
      Coil( "Unit1.Em5.ControlNodes".cmNgAndManualInputVibrator1OnOff.commands.commandWorkPos )
   END_RUNG
   // the same network as SCL:
   "Unit1.Em5.ControlNodes".cm.Interlock.ngAndManualInputVibrator1.work := #TRUE;
   "Unit1.Em5.ControlNodes".cmNgAndManualInputVibrator1OnOff.commands.commandWorkPos := NOT (NOT "Unit1.Em5.ControlNodes".ManualInput."step".action[231]);
END_REGION

REGION Network 80: Call CM NG & Manual Input Vibrator1 On/Off (LBC_TwoWayActuator)
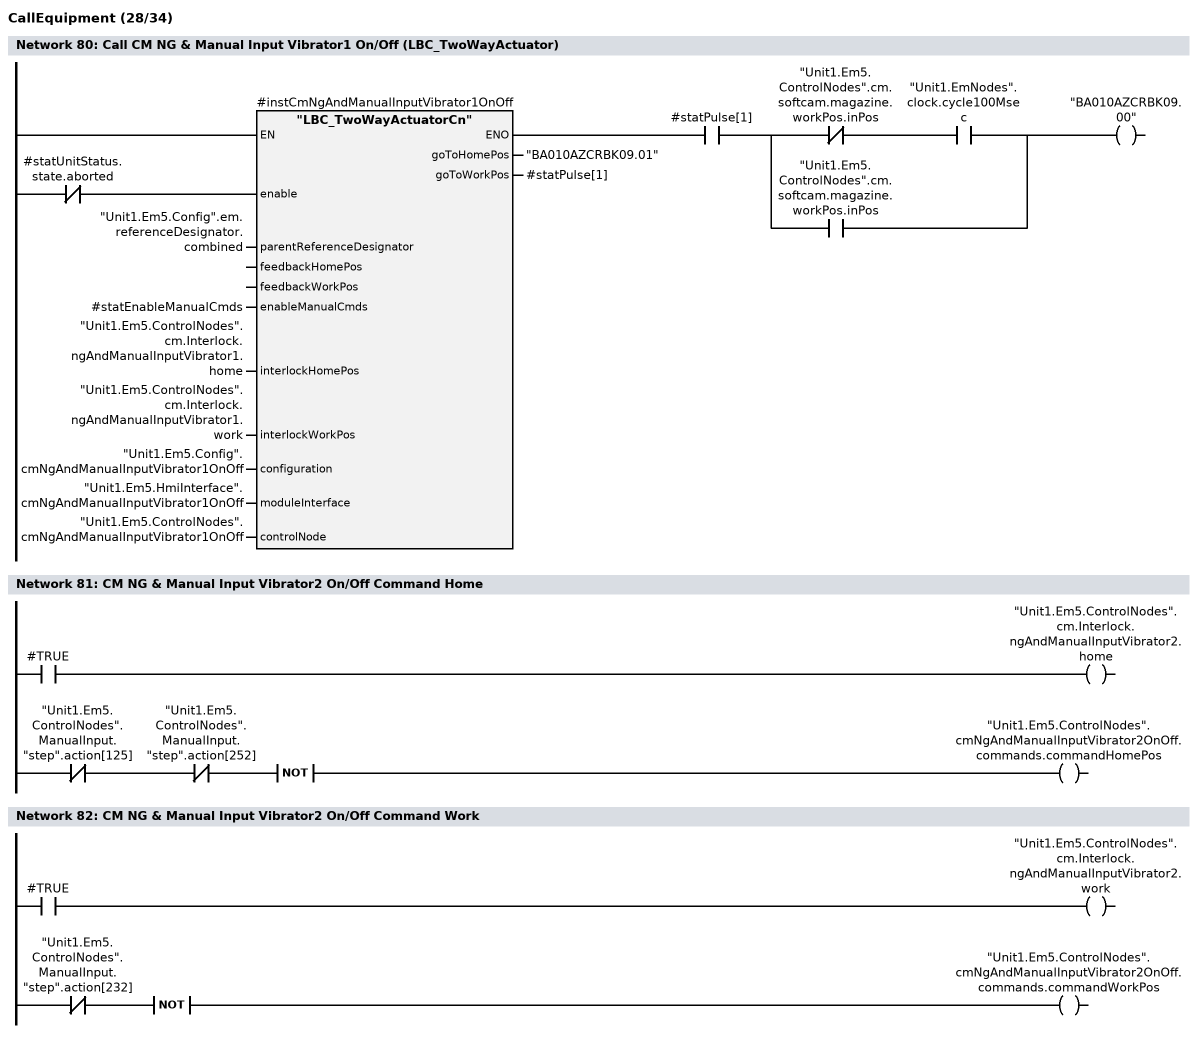
   RUNG wire#powerrail
      #instCmNgAndManualInputVibrator1OnOff(enable := wire#w1, parentReferenceDesignator := "Unit1.Em5.Config".em.referenceDesignator.combined, feedbackHomePos :=, feedbackWorkPos :=, enableManualCmds := #statEnableManualCmds, interlockHomePos := "Unit1.Em5.ControlNodes".cm.Interlock.ngAndManualInputVibrator1.home, interlockWorkPos := "Unit1.Em5.ControlNodes".cm.Interlock.ngAndManualInputVibrator1.work, configuration := "Unit1.Em5.Config".cmNgAndManualInputVibrator1OnOff, moduleInterface := "Unit1.Em5.HmiInterface".cmNgAndManualInputVibrator1OnOff, controlNode := "Unit1.Em5.ControlNodes".cmNgAndManualInputVibrator1OnOff, goToHomePos => "BA010AZCRBK09.01", goToWorkPos => #statPulse[1])
      Contact( #statPulse[1] )
      wire#w2
      I_Contact( "Unit1.Em5.ControlNodes".cm.softcam.magazine.workPos.inPos )
      Contact( "Unit1.EmNodes".clock.cycle100Msec )
      wire#w3
      Coil( "BA010AZCRBK09.00" )
   END_RUNG
   RUNG wire#powerrail
      I_Contact( #statUnitStatus.state.aborted )
   END_RUNG wire#w1
   RUNG wire#w2
      Contact( "Unit1.Em5.ControlNodes".cm.softcam.magazine.workPos.inPos )
   END_RUNG wire#w3
   // the same network as SCL:
   #instCmNgAndManualInputVibrator1OnOff(enable := NOT #statUnitStatus.state.aborted,   // "LBC_TwoWayActuatorCn"
                           parentReferenceDesignator := "Unit1.Em5.Config".em.referenceDesignator.combined,
                           enableManualCmds := #statEnableManualCmds,
                           interlockHomePos := "Unit1.Em5.ControlNodes".cm.Interlock.ngAndManualInputVibrator1.home,
                           interlockWorkPos := "Unit1.Em5.ControlNodes".cm.Interlock.ngAndManualInputVibrator1.work,
                           configuration := "Unit1.Em5.Config".cmNgAndManualInputVibrator1OnOff,
                           moduleInterface := "Unit1.Em5.HmiInterface".cmNgAndManualInputVibrator1OnOff,
                           controlNode := "Unit1.Em5.ControlNodes".cmNgAndManualInputVibrator1OnOff,
                           goToHomePos => "BA010AZCRBK09.01",
                           goToWorkPos => #statPulse[1],
                           ENO => #_w1);
   "BA010AZCRBK09.00" := #_w1 AND #statPulse[1] AND ((NOT "Unit1.Em5.ControlNodes".cm.softcam.magazine.workPos.inPos AND "Unit1.EmNodes".clock.cycle100Msec) OR "Unit1.Em5.ControlNodes".cm.softcam.magazine.workPos.inPos);
END_REGION

REGION Network 81: CM NG & Manual Input Vibrator2 On/Off Command Home
   RUNG wire#powerrail
      Contact( #TRUE )
      Coil( "Unit1.Em5.ControlNodes".cm.Interlock.ngAndManualInputVibrator2.home )
   END_RUNG
   RUNG wire#powerrail
      I_Contact( "Unit1.Em5.ControlNodes".ManualInput."step".action[125] )
      I_Contact( "Unit1.Em5.ControlNodes".ManualInput."step".action[252] )
      Not()
      Coil( "Unit1.Em5.ControlNodes".cmNgAndManualInputVibrator2OnOff.commands.commandHomePos )
   END_RUNG
   // the same network as SCL:
   "Unit1.Em5.ControlNodes".cm.Interlock.ngAndManualInputVibrator2.home := #TRUE;
   "Unit1.Em5.ControlNodes".cmNgAndManualInputVibrator2OnOff.commands.commandHomePos := NOT (NOT "Unit1.Em5.ControlNodes".ManualInput."step".action[125] AND NOT "Unit1.Em5.ControlNodes".ManualInput."step".action[252]);
END_REGION

REGION Network 82: CM NG & Manual Input Vibrator2 On/Off Command Work
   RUNG wire#powerrail
      Contact( #TRUE )
      Coil( "Unit1.Em5.ControlNodes".cm.Interlock.ngAndManualInputVibrator2.work )
   END_RUNG
   RUNG wire#powerrail
      I_Contact( "Unit1.Em5.ControlNodes".ManualInput."step".action[232] )
      Not()
      Coil( "Unit1.Em5.ControlNodes".cmNgAndManualInputVibrator2OnOff.commands.commandWorkPos )
   END_RUNG
   // the same network as SCL:
   "Unit1.Em5.ControlNodes".cm.Interlock.ngAndManualInputVibrator2.work := #TRUE;
   "Unit1.Em5.ControlNodes".cmNgAndManualInputVibrator2OnOff.commands.commandWorkPos := NOT (NOT "Unit1.Em5.ControlNodes".ManualInput."step".action[232]);
END_REGION

REGION Network 83: Call CM NG & Manual Input Vibrator2 On/Off (LBC_TwoWayActuator)
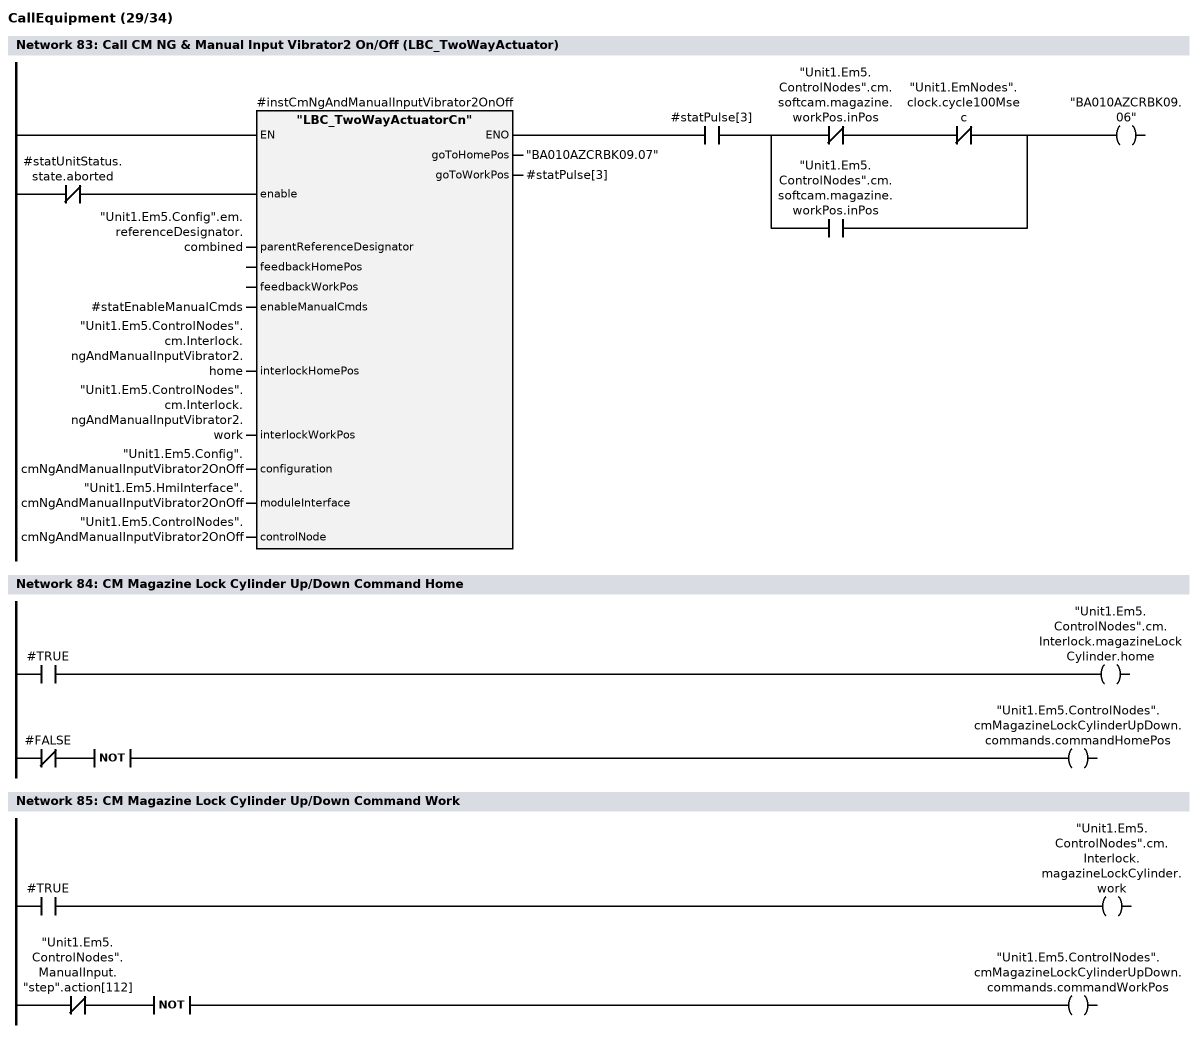
   RUNG wire#powerrail
      #instCmNgAndManualInputVibrator2OnOff(enable := wire#w1, parentReferenceDesignator := "Unit1.Em5.Config".em.referenceDesignator.combined, feedbackHomePos :=, feedbackWorkPos :=, enableManualCmds := #statEnableManualCmds, interlockHomePos := "Unit1.Em5.ControlNodes".cm.Interlock.ngAndManualInputVibrator2.home, interlockWorkPos := "Unit1.Em5.ControlNodes".cm.Interlock.ngAndManualInputVibrator2.work, configuration := "Unit1.Em5.Config".cmNgAndManualInputVibrator2OnOff, moduleInterface := "Unit1.Em5.HmiInterface".cmNgAndManualInputVibrator2OnOff, controlNode := "Unit1.Em5.ControlNodes".cmNgAndManualInputVibrator2OnOff, goToHomePos => "BA010AZCRBK09.07", goToWorkPos => #statPulse[3])
      Contact( #statPulse[3] )
      wire#w2
      I_Contact( "Unit1.Em5.ControlNodes".cm.softcam.magazine.workPos.inPos )
      I_Contact( "Unit1.EmNodes".clock.cycle100Msec )
      wire#w3
      Coil( "BA010AZCRBK09.06" )
   END_RUNG
   RUNG wire#powerrail
      I_Contact( #statUnitStatus.state.aborted )
   END_RUNG wire#w1
   RUNG wire#w2
      Contact( "Unit1.Em5.ControlNodes".cm.softcam.magazine.workPos.inPos )
   END_RUNG wire#w3
   // the same network as SCL:
   #instCmNgAndManualInputVibrator2OnOff(enable := NOT #statUnitStatus.state.aborted,   // "LBC_TwoWayActuatorCn"
                           parentReferenceDesignator := "Unit1.Em5.Config".em.referenceDesignator.combined,
                           enableManualCmds := #statEnableManualCmds,
                           interlockHomePos := "Unit1.Em5.ControlNodes".cm.Interlock.ngAndManualInputVibrator2.home,
                           interlockWorkPos := "Unit1.Em5.ControlNodes".cm.Interlock.ngAndManualInputVibrator2.work,
                           configuration := "Unit1.Em5.Config".cmNgAndManualInputVibrator2OnOff,
                           moduleInterface := "Unit1.Em5.HmiInterface".cmNgAndManualInputVibrator2OnOff,
                           controlNode := "Unit1.Em5.ControlNodes".cmNgAndManualInputVibrator2OnOff,
                           goToHomePos => "BA010AZCRBK09.07",
                           goToWorkPos => #statPulse[3],
                           ENO => #_w1);
   "BA010AZCRBK09.06" := #_w1 AND #statPulse[3] AND ((NOT "Unit1.Em5.ControlNodes".cm.softcam.magazine.workPos.inPos AND NOT "Unit1.EmNodes".clock.cycle100Msec) OR "Unit1.Em5.ControlNodes".cm.softcam.magazine.workPos.inPos);
END_REGION

REGION Network 84: CM Magazine Lock Cylinder Up/Down Command Home
   RUNG wire#powerrail
      Contact( #TRUE )
      Coil( "Unit1.Em5.ControlNodes".cm.Interlock.magazineLockCylinder.home )
   END_RUNG
   RUNG wire#powerrail
      I_Contact( #FALSE )
      Not()
      Coil( "Unit1.Em5.ControlNodes".cmMagazineLockCylinderUpDown.commands.commandHomePos )
   END_RUNG
   // the same network as SCL:
   "Unit1.Em5.ControlNodes".cm.Interlock.magazineLockCylinder.home := #TRUE;
   "Unit1.Em5.ControlNodes".cmMagazineLockCylinderUpDown.commands.commandHomePos := NOT (NOT #FALSE);
END_REGION

REGION Network 85: CM Magazine Lock Cylinder Up/Down Command Work
   RUNG wire#powerrail
      Contact( #TRUE )
      Coil( "Unit1.Em5.ControlNodes".cm.Interlock.magazineLockCylinder.work )
   END_RUNG
   RUNG wire#powerrail
      I_Contact( "Unit1.Em5.ControlNodes".ManualInput."step".action[112] )
      Not()
      Coil( "Unit1.Em5.ControlNodes".cmMagazineLockCylinderUpDown.commands.commandWorkPos )
   END_RUNG
   // the same network as SCL:
   "Unit1.Em5.ControlNodes".cm.Interlock.magazineLockCylinder.work := #TRUE;
   "Unit1.Em5.ControlNodes".cmMagazineLockCylinderUpDown.commands.commandWorkPos := NOT (NOT "Unit1.Em5.ControlNodes".ManualInput."step".action[112]);
END_REGION

REGION Network 86: Call CM Magazine Lock Cylinder Up/Down (LBC_TwoWayActuator)
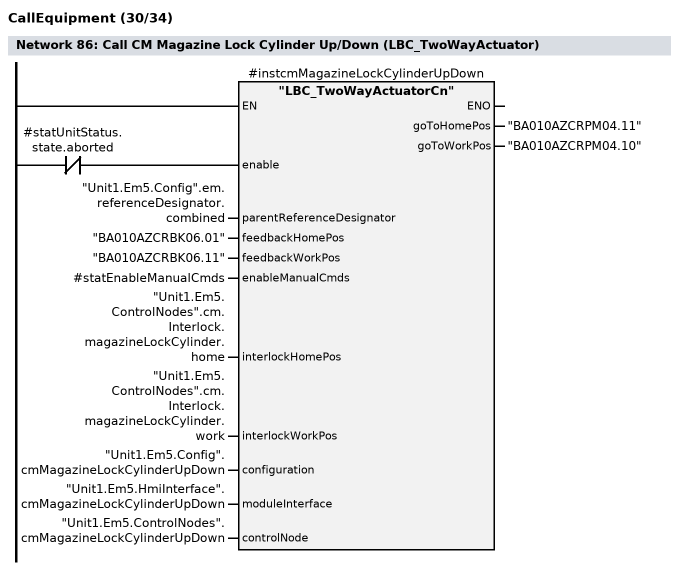
   RUNG wire#powerrail
      #instcmMagazineLockCylinderUpDown(enable := wire#w1, parentReferenceDesignator := "Unit1.Em5.Config".em.referenceDesignator.combined, feedbackHomePos := "BA010AZCRBK06.01", feedbackWorkPos := "BA010AZCRBK06.11", enableManualCmds := #statEnableManualCmds, interlockHomePos := "Unit1.Em5.ControlNodes".cm.Interlock.magazineLockCylinder.home, interlockWorkPos := "Unit1.Em5.ControlNodes".cm.Interlock.magazineLockCylinder.work, configuration := "Unit1.Em5.Config".cmMagazineLockCylinderUpDown, moduleInterface := "Unit1.Em5.HmiInterface".cmMagazineLockCylinderUpDown, controlNode := "Unit1.Em5.ControlNodes".cmMagazineLockCylinderUpDown, goToHomePos => "BA010AZCRPM04.11", goToWorkPos => "BA010AZCRPM04.10")
   END_RUNG
   RUNG wire#powerrail
      I_Contact( #statUnitStatus.state.aborted )
   END_RUNG wire#w1
   // the same network as SCL:
   #instcmMagazineLockCylinderUpDown(enable := NOT #statUnitStatus.state.aborted,   // "LBC_TwoWayActuatorCn"
                           parentReferenceDesignator := "Unit1.Em5.Config".em.referenceDesignator.combined,
                           feedbackHomePos := "BA010AZCRBK06.01",
                           feedbackWorkPos := "BA010AZCRBK06.11",
                           enableManualCmds := #statEnableManualCmds,
                           interlockHomePos := "Unit1.Em5.ControlNodes".cm.Interlock.magazineLockCylinder.home,
                           interlockWorkPos := "Unit1.Em5.ControlNodes".cm.Interlock.magazineLockCylinder.work,
                           configuration := "Unit1.Em5.Config".cmMagazineLockCylinderUpDown,
                           moduleInterface := "Unit1.Em5.HmiInterface".cmMagazineLockCylinderUpDown,
                           controlNode := "Unit1.Em5.ControlNodes".cmMagazineLockCylinderUpDown,
                           goToHomePos => "BA010AZCRPM04.11",
                           goToWorkPos => "BA010AZCRPM04.10");
END_REGION

REGION Network 87: ******************** Feedback to Unit ********************
END_REGION

REGION Network 88: Determine StateComplete (SC) in Mode Production
   // Conditions for the Equipment Modules "stateComplete" feedback to the unit. This feedback is given when the task in for the respective state is complete.
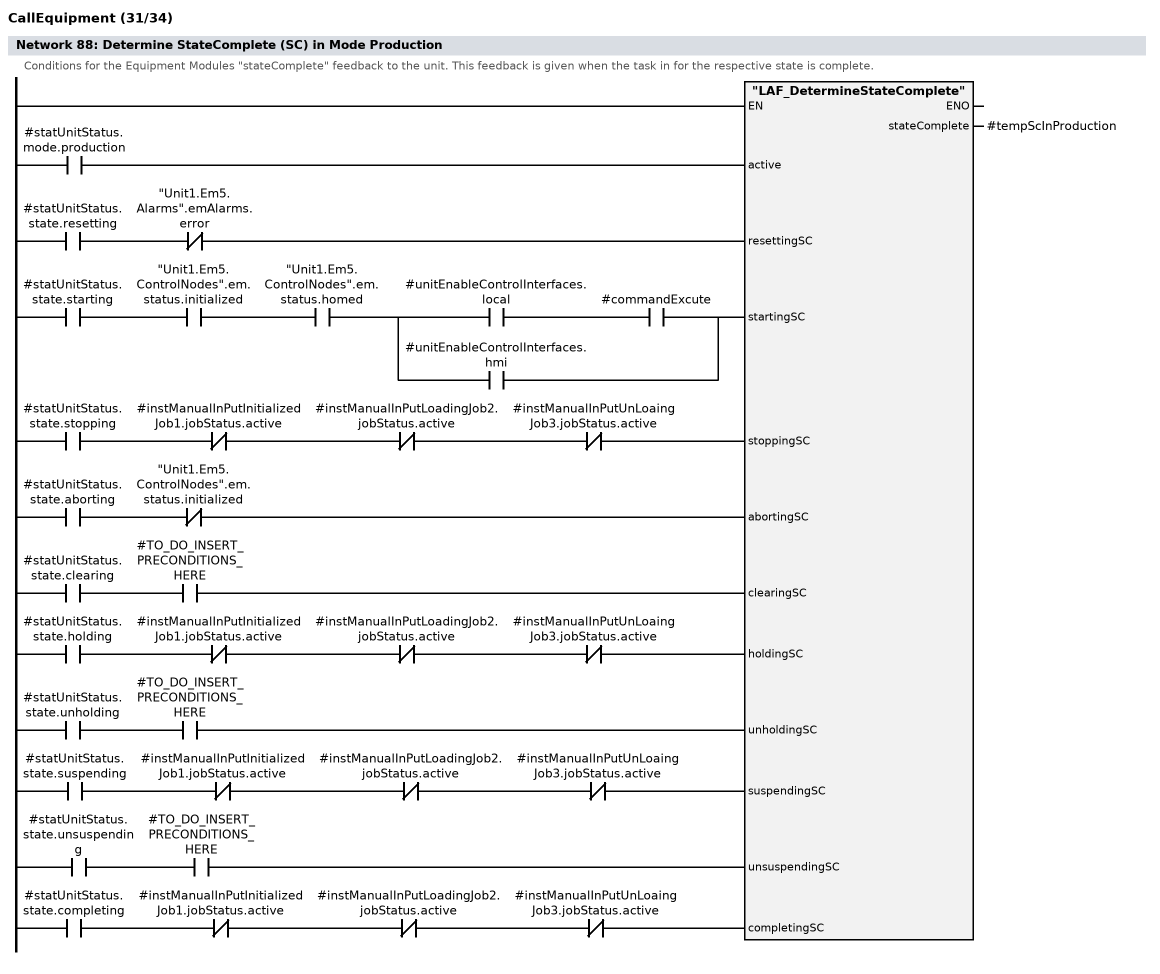
   RUNG wire#powerrail
      "LAF_DetermineStateComplete"(active := wire#w1, resettingSC := wire#w2, startingSC := wire#w4, stoppingSC := wire#w5, abortingSC := wire#w6, clearingSC := wire#w7, holdingSC := wire#w8, unholdingSC := wire#w9, suspendingSC := wire#w10, unsuspendingSC := wire#w11, completingSC := wire#w12, stateComplete => #tempScInProduction)
   END_RUNG
   RUNG wire#powerrail
      Contact( #statUnitStatus.mode.production )
   END_RUNG wire#w1
   RUNG wire#powerrail
      Contact( #statUnitStatus.state.resetting )
      I_Contact( "Unit1.Em5.Alarms".emAlarms.error )
   END_RUNG wire#w2
   RUNG wire#powerrail
      Contact( #statUnitStatus.state.starting )
      Contact( "Unit1.Em5.ControlNodes".em.status.initialized )
      Contact( "Unit1.Em5.ControlNodes".em.status.homed )
      wire#w3
      Contact( #unitEnableControlInterfaces.local )
      Contact( #commandExcute )
   END_RUNG wire#w4
   RUNG wire#w3
      Contact( #unitEnableControlInterfaces.hmi )
   END_RUNG wire#w4
   RUNG wire#powerrail
      Contact( #statUnitStatus.state.stopping )
      I_Contact( #instManualInPutInitializedJob1.jobStatus.active )
      I_Contact( #instManualInPutLoadingJob2.jobStatus.active )
      I_Contact( #instManualInPutUnLoaingJob3.jobStatus.active )
   END_RUNG wire#w5
   RUNG wire#powerrail
      Contact( #statUnitStatus.state.aborting )
      I_Contact( "Unit1.Em5.ControlNodes".em.status.initialized )
   END_RUNG wire#w6
   RUNG wire#powerrail
      Contact( #statUnitStatus.state.clearing )
      Contact( #TO_DO_INSERT_PRECONDITIONS_HERE )
   END_RUNG wire#w7
   RUNG wire#powerrail
      Contact( #statUnitStatus.state.holding )
      I_Contact( #instManualInPutInitializedJob1.jobStatus.active )
      I_Contact( #instManualInPutLoadingJob2.jobStatus.active )
      I_Contact( #instManualInPutUnLoaingJob3.jobStatus.active )
   END_RUNG wire#w8
   RUNG wire#powerrail
      Contact( #statUnitStatus.state.unholding )
      Contact( #TO_DO_INSERT_PRECONDITIONS_HERE )
   END_RUNG wire#w9
   RUNG wire#powerrail
      Contact( #statUnitStatus.state.suspending )
      I_Contact( #instManualInPutInitializedJob1.jobStatus.active )
      I_Contact( #instManualInPutLoadingJob2.jobStatus.active )
      I_Contact( #instManualInPutUnLoaingJob3.jobStatus.active )
   END_RUNG wire#w10
   RUNG wire#powerrail
      Contact( #statUnitStatus.state.unsuspending )
      Contact( #TO_DO_INSERT_PRECONDITIONS_HERE )
   END_RUNG wire#w11
   RUNG wire#powerrail
      Contact( #statUnitStatus.state.completing )
      I_Contact( #instManualInPutInitializedJob1.jobStatus.active )
      I_Contact( #instManualInPutLoadingJob2.jobStatus.active )
      I_Contact( #instManualInPutUnLoaingJob3.jobStatus.active )
   END_RUNG wire#w12
   // the same network as SCL:
   "LAF_DetermineStateComplete"(active := #statUnitStatus.mode.production,
                           resettingSC := #statUnitStatus.state.resetting AND NOT "Unit1.Em5.Alarms".emAlarms.error,
                           startingSC := #statUnitStatus.state.starting AND "Unit1.Em5.ControlNodes".em.status.initialized AND "Unit1.Em5.ControlNodes".em.status.homed AND ((#unitEnableControlInterfaces.local AND #commandExcute) OR #unitEnableControlInterfaces.hmi),
                           stoppingSC := #statUnitStatus.state.stopping AND NOT #instManualInPutInitializedJob1.jobStatus.active AND NOT #instManualInPutLoadingJob2.jobStatus.active AND NOT #instManualInPutUnLoaingJob3.jobStatus.active,
                           abortingSC := #statUnitStatus.state.aborting AND NOT "Unit1.Em5.ControlNodes".em.status.initialized,
                           clearingSC := #statUnitStatus.state.clearing AND #TO_DO_INSERT_PRECONDITIONS_HERE,
                           holdingSC := #statUnitStatus.state.holding AND NOT #instManualInPutInitializedJob1.jobStatus.active AND NOT #instManualInPutLoadingJob2.jobStatus.active AND NOT #instManualInPutUnLoaingJob3.jobStatus.active,
                           unholdingSC := #statUnitStatus.state.unholding AND #TO_DO_INSERT_PRECONDITIONS_HERE,
                           suspendingSC := #statUnitStatus.state.suspending AND NOT #instManualInPutInitializedJob1.jobStatus.active AND NOT #instManualInPutLoadingJob2.jobStatus.active AND NOT #instManualInPutUnLoaingJob3.jobStatus.active,
                           unsuspendingSC := #statUnitStatus.state.unsuspending AND #TO_DO_INSERT_PRECONDITIONS_HERE,
                           completingSC := #statUnitStatus.state.completing AND NOT #instManualInPutInitializedJob1.jobStatus.active AND NOT #instManualInPutLoadingJob2.jobStatus.active AND NOT #instManualInPutUnLoaingJob3.jobStatus.active,
                           stateComplete => #tempScInProduction);
END_REGION

REGION Network 89: Determine StateComplete (SC) in Mode Maintenance/Manual
   // Conditions for the Equipment Modules "stateComplete" feedback to the unit. This feedback is given when the task in for the respective state is complete.
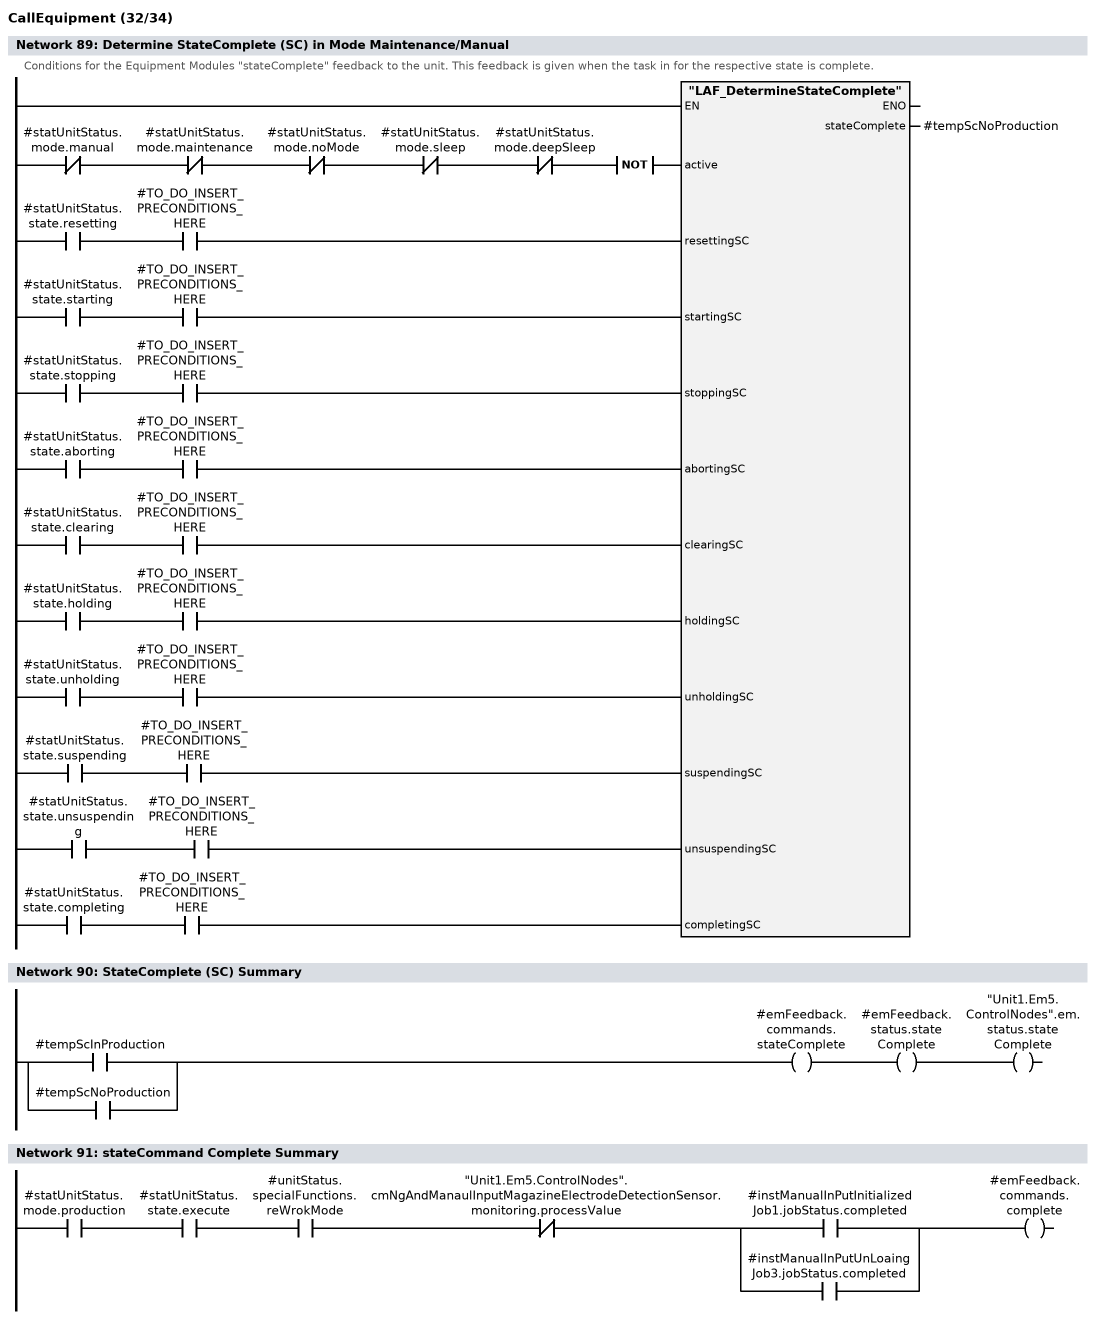
   RUNG wire#powerrail
      "LAF_DetermineStateComplete"(active := wire#w1, resettingSC := wire#w2, startingSC := wire#w3, stoppingSC := wire#w4, abortingSC := wire#w5, clearingSC := wire#w6, holdingSC := wire#w7, unholdingSC := wire#w8, suspendingSC := wire#w9, unsuspendingSC := wire#w10, completingSC := wire#w11, stateComplete => #tempScNoProduction)
   END_RUNG
   RUNG wire#powerrail
      I_Contact( #statUnitStatus.mode.manual )
      I_Contact( #statUnitStatus.mode.maintenance )
      I_Contact( #statUnitStatus.mode.noMode )
      I_Contact( #statUnitStatus.mode.sleep )
      I_Contact( #statUnitStatus.mode.deepSleep )
      Not()
   END_RUNG wire#w1
   RUNG wire#powerrail
      Contact( #statUnitStatus.state.resetting )
      Contact( #TO_DO_INSERT_PRECONDITIONS_HERE )
   END_RUNG wire#w2
   RUNG wire#powerrail
      Contact( #statUnitStatus.state.starting )
      Contact( #TO_DO_INSERT_PRECONDITIONS_HERE )
   END_RUNG wire#w3
   RUNG wire#powerrail
      Contact( #statUnitStatus.state.stopping )
      Contact( #TO_DO_INSERT_PRECONDITIONS_HERE )
   END_RUNG wire#w4
   RUNG wire#powerrail
      Contact( #statUnitStatus.state.aborting )
      Contact( #TO_DO_INSERT_PRECONDITIONS_HERE )
   END_RUNG wire#w5
   RUNG wire#powerrail
      Contact( #statUnitStatus.state.clearing )
      Contact( #TO_DO_INSERT_PRECONDITIONS_HERE )
   END_RUNG wire#w6
   RUNG wire#powerrail
      Contact( #statUnitStatus.state.holding )
      Contact( #TO_DO_INSERT_PRECONDITIONS_HERE )
   END_RUNG wire#w7
   RUNG wire#powerrail
      Contact( #statUnitStatus.state.unholding )
      Contact( #TO_DO_INSERT_PRECONDITIONS_HERE )
   END_RUNG wire#w8
   RUNG wire#powerrail
      Contact( #statUnitStatus.state.suspending )
      Contact( #TO_DO_INSERT_PRECONDITIONS_HERE )
   END_RUNG wire#w9
   RUNG wire#powerrail
      Contact( #statUnitStatus.state.unsuspending )
      Contact( #TO_DO_INSERT_PRECONDITIONS_HERE )
   END_RUNG wire#w10
   RUNG wire#powerrail
      Contact( #statUnitStatus.state.completing )
      Contact( #TO_DO_INSERT_PRECONDITIONS_HERE )
   END_RUNG wire#w11
   // the same network as SCL:
   "LAF_DetermineStateComplete"(active := NOT (NOT #statUnitStatus.mode.manual AND NOT #statUnitStatus.mode.maintenance AND NOT #statUnitStatus.mode.noMode AND NOT #statUnitStatus.mode.sleep AND NOT #statUnitStatus.mode.deepSleep),
                           resettingSC := #statUnitStatus.state.resetting AND #TO_DO_INSERT_PRECONDITIONS_HERE,
                           startingSC := #statUnitStatus.state.starting AND #TO_DO_INSERT_PRECONDITIONS_HERE,
                           stoppingSC := #statUnitStatus.state.stopping AND #TO_DO_INSERT_PRECONDITIONS_HERE,
                           abortingSC := #statUnitStatus.state.aborting AND #TO_DO_INSERT_PRECONDITIONS_HERE,
                           clearingSC := #statUnitStatus.state.clearing AND #TO_DO_INSERT_PRECONDITIONS_HERE,
                           holdingSC := #statUnitStatus.state.holding AND #TO_DO_INSERT_PRECONDITIONS_HERE,
                           unholdingSC := #statUnitStatus.state.unholding AND #TO_DO_INSERT_PRECONDITIONS_HERE,
                           suspendingSC := #statUnitStatus.state.suspending AND #TO_DO_INSERT_PRECONDITIONS_HERE,
                           unsuspendingSC := #statUnitStatus.state.unsuspending AND #TO_DO_INSERT_PRECONDITIONS_HERE,
                           completingSC := #statUnitStatus.state.completing AND #TO_DO_INSERT_PRECONDITIONS_HERE,
                           stateComplete => #tempScNoProduction);
END_REGION

REGION Network 90: StateComplete (SC) Summary
   RUNG wire#powerrail
      Contact( #tempScInProduction )
      wire#w1
      Coil( #emFeedback.commands.stateComplete )
      Coil( #emFeedback.status.stateComplete )
      Coil( "Unit1.Em5.ControlNodes".em.status.stateComplete )
   END_RUNG
   RUNG wire#powerrail
      Contact( #tempScNoProduction )
   END_RUNG wire#w1
   // the same network as SCL:
   #emFeedback.commands.stateComplete := #tempScInProduction OR #tempScNoProduction;
   #emFeedback.status.stateComplete := #emFeedback.commands.stateComplete;
   "Unit1.Em5.ControlNodes".em.status.stateComplete := #emFeedback.commands.stateComplete;
END_REGION

REGION Network 91: stateCommand Complete Summary
   RUNG wire#powerrail
      Contact( #statUnitStatus.mode.production )
      Contact( #statUnitStatus.state.execute )
      Contact( #unitStatus.specialFunctions.reWrokMode )
      I_Contact( "Unit1.Em5.ControlNodes".cmNgAndManaulInputMagazineElectrodeDetectionSensor.monitoring.processValue )
      wire#w1
      Contact( #instManualInPutInitializedJob1.jobStatus.completed )
      wire#w2
      Coil( #emFeedback.commands.complete )
   END_RUNG
   RUNG wire#w1
      Contact( #instManualInPutUnLoaingJob3.jobStatus.completed )
   END_RUNG wire#w2
   // the same network as SCL:
   #emFeedback.commands.complete := #statUnitStatus.mode.production AND #statUnitStatus.state.execute AND #unitStatus.specialFunctions.reWrokMode AND NOT "Unit1.Em5.ControlNodes".cmNgAndManaulInputMagazineElectrodeDetectionSensor.monitoring.processValue AND (#instManualInPutInitializedJob1.jobStatus.completed OR #instManualInPutUnLoaingJob3.jobStatus.completed);
END_REGION

REGION Network 92: status safeState Summary
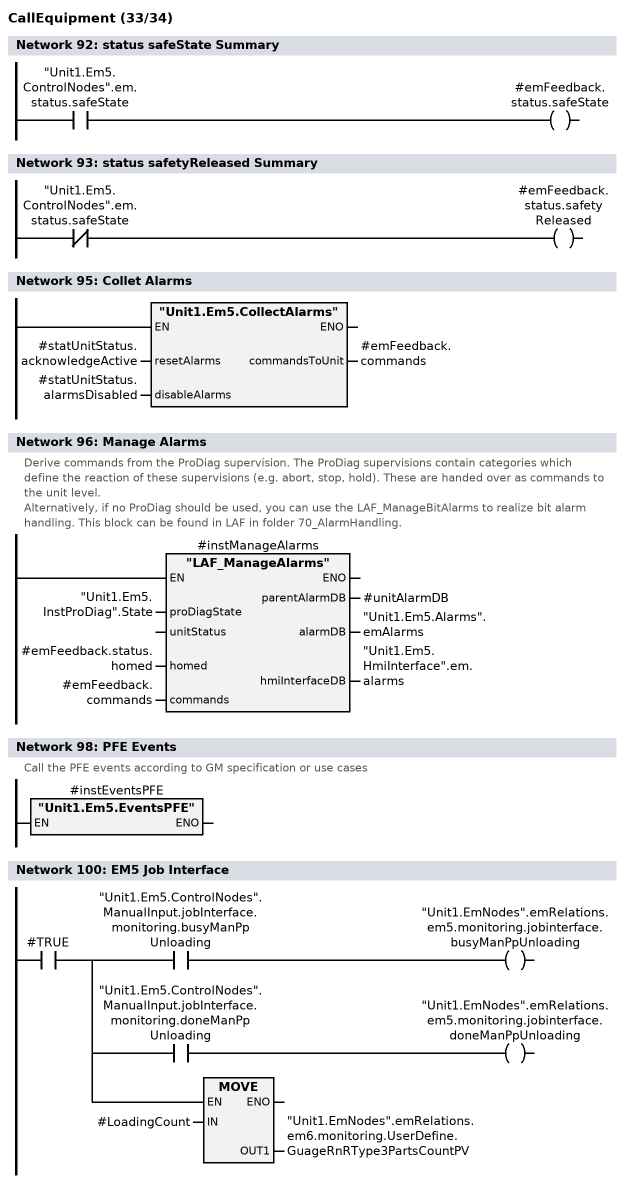
   RUNG wire#powerrail
      Contact( "Unit1.Em5.ControlNodes".em.status.safeState )
      Coil( #emFeedback.status.safeState )
   END_RUNG
   // the same network as SCL:
   #emFeedback.status.safeState := "Unit1.Em5.ControlNodes".em.status.safeState;
END_REGION

REGION Network 93: status safetyReleased Summary
   RUNG wire#powerrail
      I_Contact( "Unit1.Em5.ControlNodes".em.status.safeState )
      Coil( #emFeedback.status.safetyReleased )
   END_RUNG
   // the same network as SCL:
   #emFeedback.status.safetyReleased := NOT "Unit1.Em5.ControlNodes".em.status.safeState;
END_REGION

REGION Network 94: ******************** Alarms ********************
END_REGION

REGION Network 95: Collet Alarms
   RUNG wire#powerrail
      "Unit1.Em5.CollectAlarms"(resetAlarms := #statUnitStatus.acknowledgeActive, disableAlarms := #statUnitStatus.alarmsDisabled, commandsToUnit => #emFeedback.commands)
   END_RUNG
   // the same network as SCL:
   "Unit1.Em5.CollectAlarms"(resetAlarms := #statUnitStatus.acknowledgeActive,
                           disableAlarms := #statUnitStatus.alarmsDisabled,
                           commandsToUnit => #emFeedback.commands);
END_REGION

REGION Network 96: Manage Alarms
   // Derive commands from the ProDiag supervision. The ProDiag supervisions contain categories which define the reaction of these supervisions (e.g. abort, stop, hold). These are handed over as commands to the unit level.
   // Alternatively, if no ProDiag should be used, you can use the LAF_ManageBitAlarms to realize bit alarm handling. This block can be found in LAF in folder 70_AlarmHandling.
   RUNG wire#powerrail
      #instManageAlarms(proDiagState := "Unit1.Em5.InstProDiag".State, unitStatus :=, homed := #emFeedback.status.homed, commands := #emFeedback.commands, parentAlarmDB => #unitAlarmDB, alarmDB => "Unit1.Em5.Alarms".emAlarms, hmiInterfaceDB => "Unit1.Em5.HmiInterface".em.alarms)
   END_RUNG
   // the same network as SCL:
   #instManageAlarms(proDiagState := "Unit1.Em5.InstProDiag".State,   // "LAF_ManageAlarms"
                     homed := #emFeedback.status.homed,
                     commands := #emFeedback.commands,
                     parentAlarmDB => #unitAlarmDB,
                     alarmDB => "Unit1.Em5.Alarms".emAlarms,
                     hmiInterfaceDB => "Unit1.Em5.HmiInterface".em.alarms);
END_REGION

REGION Network 97: ******************** PFE Events ********************
END_REGION

REGION Network 98: PFE Events
   // Call the PFE events according to GM specification or use cases
   RUNG wire#powerrail
      #instEventsPFE()
   END_RUNG
   // the same network as SCL:
   #instEventsPFE();   // "Unit1.Em5.EventsPFE"
END_REGION

REGION Network 99: ******************** EM Relations Output ********************
END_REGION

REGION Network 100: EM5 Job Interface
   RUNG wire#powerrail
      Contact( #TRUE )
      wire#w1
      Contact( "Unit1.Em5.ControlNodes".ManualInput.jobInterface.monitoring.busyManPpUnloading )
      Coil( "Unit1.EmNodes".emRelations.em5.monitoring.jobinterface.busyManPpUnloading )
   END_RUNG
   RUNG wire#w1
      Contact( "Unit1.Em5.ControlNodes".ManualInput.jobInterface.monitoring.doneManPpUnloading )
      Coil( "Unit1.EmNodes".emRelations.em5.monitoring.jobinterface.doneManPpUnloading )
   END_RUNG
   RUNG wire#w1
      Move(in := #LoadingCount, out1 => "Unit1.EmNodes".emRelations.em6.monitoring.UserDefine.GuageRnRType3PartsCountPV)
   END_RUNG
   // the same network as SCL:
   "Unit1.EmNodes".emRelations.em5.monitoring.jobinterface.busyManPpUnloading := #TRUE AND "Unit1.Em5.ControlNodes".ManualInput.jobInterface.monitoring.busyManPpUnloading;
   "Unit1.EmNodes".emRelations.em5.monitoring.jobinterface.doneManPpUnloading := #TRUE AND "Unit1.Em5.ControlNodes".ManualInput.jobInterface.monitoring.doneManPpUnloading;
   IF #TRUE THEN
       "Unit1.EmNodes".emRelations.em6.monitoring.UserDefine.GuageRnRType3PartsCountPV := #LoadingCount;
   END_IF;
END_REGION

REGION Network 101: EM5 cmStatus
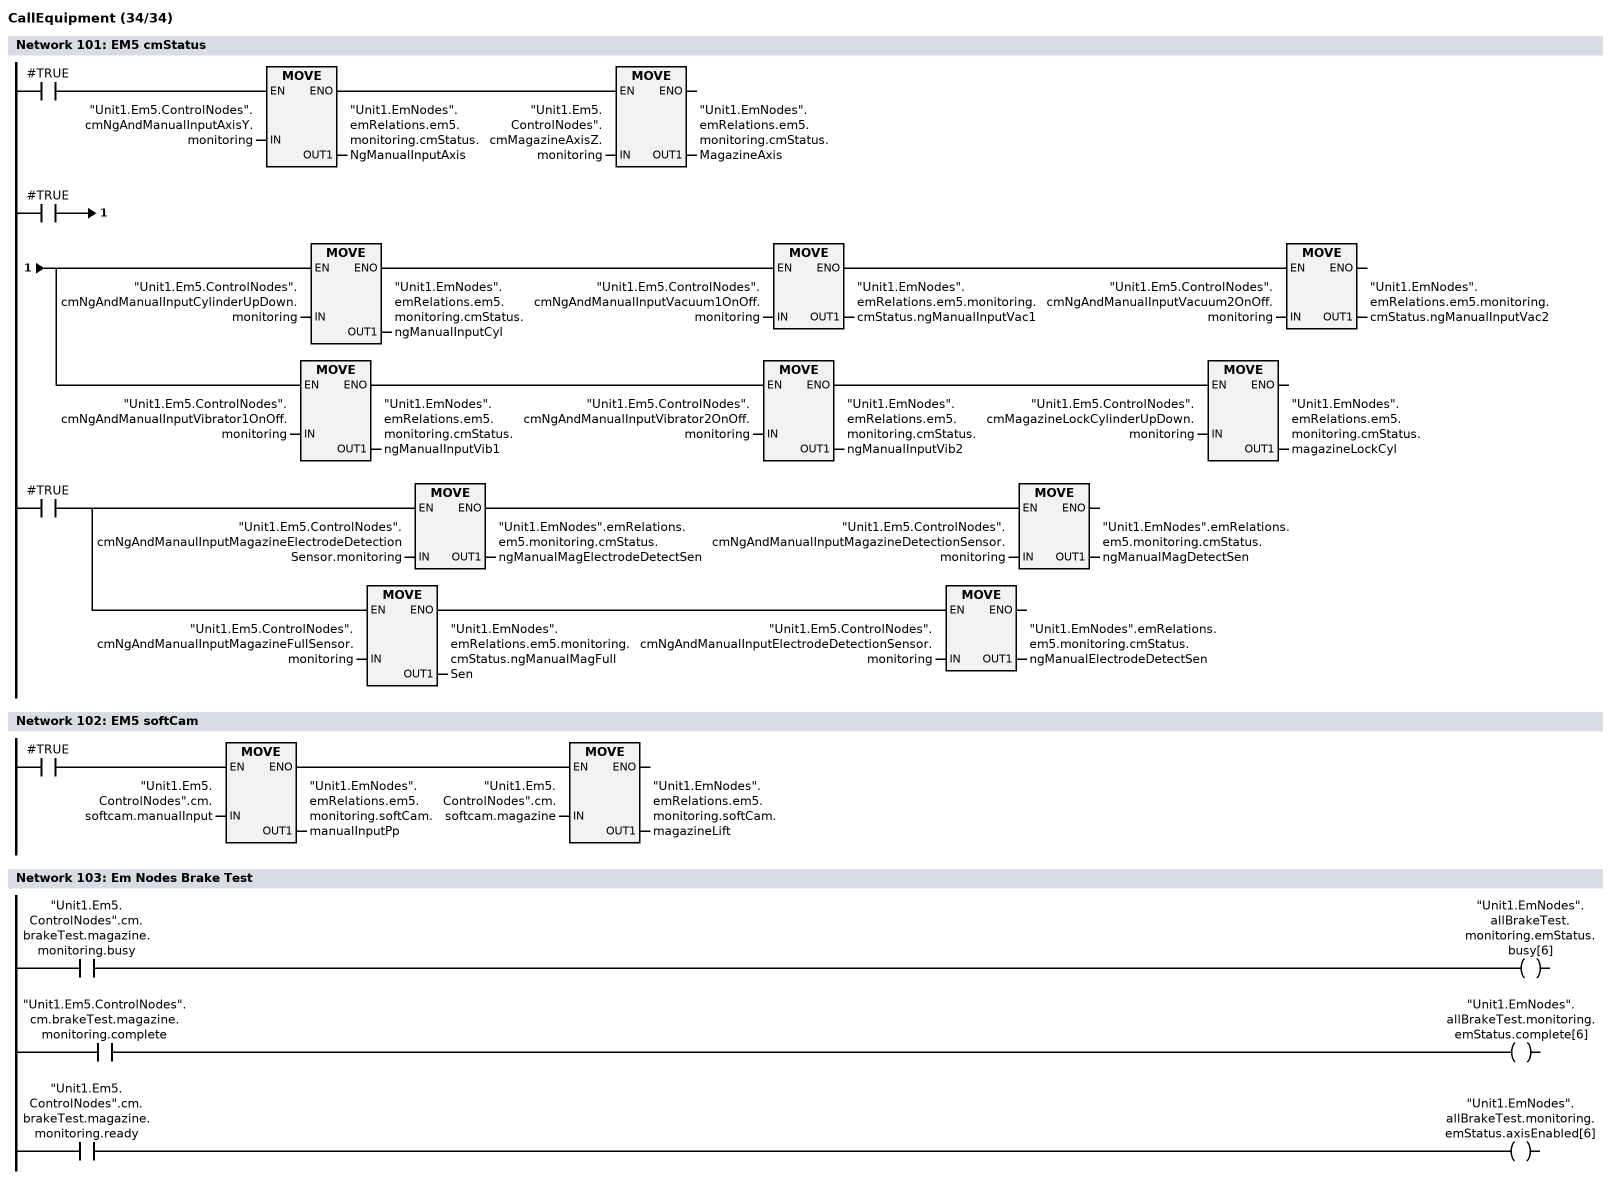
   RUNG wire#powerrail
      Contact( #TRUE )
      Move(in := "Unit1.Em5.ControlNodes".cmNgAndManualInputAxisY.monitoring, out1 => "Unit1.EmNodes".emRelations.em5.monitoring.cmStatus.NgManualInputAxis)
      Move(in := "Unit1.Em5.ControlNodes".cmMagazineAxisZ.monitoring, out1 => "Unit1.EmNodes".emRelations.em5.monitoring.cmStatus.MagazineAxis)
   END_RUNG
   RUNG wire#powerrail
      Contact( #TRUE )
      wire#w1
      Move(in := "Unit1.Em5.ControlNodes".cmNgAndManualInputCylinderUpDown.monitoring, out1 => "Unit1.EmNodes".emRelations.em5.monitoring.cmStatus.ngManualInputCyl)
      Move(in := "Unit1.Em5.ControlNodes".cmNgAndManualInputVacuum1OnOff.monitoring, out1 => "Unit1.EmNodes".emRelations.em5.monitoring.cmStatus.ngManualInputVac1)
      Move(in := "Unit1.Em5.ControlNodes".cmNgAndManualInputVacuum2OnOff.monitoring, out1 => "Unit1.EmNodes".emRelations.em5.monitoring.cmStatus.ngManualInputVac2)
   END_RUNG
   RUNG wire#w1
      Move(in := "Unit1.Em5.ControlNodes".cmNgAndManualInputVibrator1OnOff.monitoring, out1 => "Unit1.EmNodes".emRelations.em5.monitoring.cmStatus.ngManualInputVib1)
      Move(in := "Unit1.Em5.ControlNodes".cmNgAndManualInputVibrator2OnOff.monitoring, out1 => "Unit1.EmNodes".emRelations.em5.monitoring.cmStatus.ngManualInputVib2)
      Move(in := "Unit1.Em5.ControlNodes".cmMagazineLockCylinderUpDown.monitoring, out1 => "Unit1.EmNodes".emRelations.em5.monitoring.cmStatus.magazineLockCyl)
   END_RUNG
   RUNG wire#powerrail
      Contact( #TRUE )
      wire#w2
      Move(in := "Unit1.Em5.ControlNodes".cmNgAndManaulInputMagazineElectrodeDetectionSensor.monitoring, out1 => "Unit1.EmNodes".emRelations.em5.monitoring.cmStatus.ngManualMagElectrodeDetectSen)
      Move(in := "Unit1.Em5.ControlNodes".cmNgAndManualInputMagazineDetectionSensor.monitoring, out1 => "Unit1.EmNodes".emRelations.em5.monitoring.cmStatus.ngManualMagDetectSen)
   END_RUNG
   RUNG wire#w2
      Move(in := "Unit1.Em5.ControlNodes".cmNgAndManualInputMagazineFullSensor.monitoring, out1 => "Unit1.EmNodes".emRelations.em5.monitoring.cmStatus.ngManualMagFullSen)
      Move(in := "Unit1.Em5.ControlNodes".cmNgAndManualInputElectrodeDetectionSensor.monitoring, out1 => "Unit1.EmNodes".emRelations.em5.monitoring.cmStatus.ngManualElectrodeDetectSen)
   END_RUNG
   // the same network as SCL:
   IF #TRUE THEN
       "Unit1.EmNodes".emRelations.em5.monitoring.cmStatus.NgManualInputAxis := "Unit1.Em5.ControlNodes".cmNgAndManualInputAxisY.monitoring;
       "Unit1.EmNodes".emRelations.em5.monitoring.cmStatus.MagazineAxis := "Unit1.Em5.ControlNodes".cmMagazineAxisZ.monitoring;
       "Unit1.EmNodes".emRelations.em5.monitoring.cmStatus.ngManualInputCyl := "Unit1.Em5.ControlNodes".cmNgAndManualInputCylinderUpDown.monitoring;
       "Unit1.EmNodes".emRelations.em5.monitoring.cmStatus.ngManualInputVac1 := "Unit1.Em5.ControlNodes".cmNgAndManualInputVacuum1OnOff.monitoring;
       "Unit1.EmNodes".emRelations.em5.monitoring.cmStatus.ngManualInputVac2 := "Unit1.Em5.ControlNodes".cmNgAndManualInputVacuum2OnOff.monitoring;
       "Unit1.EmNodes".emRelations.em5.monitoring.cmStatus.ngManualInputVib1 := "Unit1.Em5.ControlNodes".cmNgAndManualInputVibrator1OnOff.monitoring;
       "Unit1.EmNodes".emRelations.em5.monitoring.cmStatus.ngManualInputVib2 := "Unit1.Em5.ControlNodes".cmNgAndManualInputVibrator2OnOff.monitoring;
       "Unit1.EmNodes".emRelations.em5.monitoring.cmStatus.magazineLockCyl := "Unit1.Em5.ControlNodes".cmMagazineLockCylinderUpDown.monitoring;
       "Unit1.EmNodes".emRelations.em5.monitoring.cmStatus.ngManualMagElectrodeDetectSen := "Unit1.Em5.ControlNodes".cmNgAndManaulInputMagazineElectrodeDetectionSensor.monitoring;
       "Unit1.EmNodes".emRelations.em5.monitoring.cmStatus.ngManualMagDetectSen := "Unit1.Em5.ControlNodes".cmNgAndManualInputMagazineDetectionSensor.monitoring;
       "Unit1.EmNodes".emRelations.em5.monitoring.cmStatus.ngManualMagFullSen := "Unit1.Em5.ControlNodes".cmNgAndManualInputMagazineFullSensor.monitoring;
       "Unit1.EmNodes".emRelations.em5.monitoring.cmStatus.ngManualElectrodeDetectSen := "Unit1.Em5.ControlNodes".cmNgAndManualInputElectrodeDetectionSensor.monitoring;
   END_IF;
END_REGION

REGION Network 102: EM5 softCam
   RUNG wire#powerrail
      Contact( #TRUE )
      Move(in := "Unit1.Em5.ControlNodes".cm.softcam.manualInput, out1 => "Unit1.EmNodes".emRelations.em5.monitoring.softCam.manualInputPp)
      Move(in := "Unit1.Em5.ControlNodes".cm.softcam.magazine, out1 => "Unit1.EmNodes".emRelations.em5.monitoring.softCam.magazineLift)
   END_RUNG
   // the same network as SCL:
   IF #TRUE THEN
       "Unit1.EmNodes".emRelations.em5.monitoring.softCam.manualInputPp := "Unit1.Em5.ControlNodes".cm.softcam.manualInput;
       "Unit1.EmNodes".emRelations.em5.monitoring.softCam.magazineLift := "Unit1.Em5.ControlNodes".cm.softcam.magazine;
   END_IF;
END_REGION

REGION Network 103: Em Nodes Brake Test
   RUNG wire#powerrail
      Contact( "Unit1.Em5.ControlNodes".cm.brakeTest.magazine.monitoring.busy )
      Coil( "Unit1.EmNodes".allBrakeTest.monitoring.emStatus.busy[6] )
   END_RUNG
   RUNG wire#powerrail
      Contact( "Unit1.Em5.ControlNodes".cm.brakeTest.magazine.monitoring.complete )
      Coil( "Unit1.EmNodes".allBrakeTest.monitoring.emStatus.complete[6] )
   END_RUNG
   RUNG wire#powerrail
      Contact( "Unit1.Em5.ControlNodes".cm.brakeTest.magazine.monitoring.ready )
      Coil( "Unit1.EmNodes".allBrakeTest.monitoring.emStatus.axisEnabled[6] )
   END_RUNG
   // the same network as SCL:
   "Unit1.EmNodes".allBrakeTest.monitoring.emStatus.busy[6] := "Unit1.Em5.ControlNodes".cm.brakeTest.magazine.monitoring.busy;
   "Unit1.EmNodes".allBrakeTest.monitoring.emStatus.complete[6] := "Unit1.Em5.ControlNodes".cm.brakeTest.magazine.monitoring.complete;
   "Unit1.EmNodes".allBrakeTest.monitoring.emStatus.axisEnabled[6] := "Unit1.Em5.ControlNodes".cm.brakeTest.magazine.monitoring.ready;
END_REGION
END_FUNCTION_BLOCK
